SPLINE
SPL {X  -120.253, Y  +789.426, Z    +0.000, E1   -51.165, E3 +212498.946}
SPL {X  -143.101, Y  +758.939, Z    +0.000, E1   -44.365, E3 +212513.054}
SPL {X  -158.740, Y  +722.846, Z    +0.000, E1   -30.140, E3 +212511.093}
SPL {X  -163.639, Y  +701.236, Z    +0.000, E1   -18.901, E3 +212513.231}
SPL {X  -165.058, Y  +689.494, Z    +0.000, E1   -11.557, E3 +212512.047}
SPL {X  -165.574, Y  +680.514, Z    +0.000, E1    -5.500, E3 +212511.291}
SPL {X  -165.650, Y  +673.883, Z    +0.000, E1    -0.454, E3 +212510.302}
SPL {X  -165.650, Y  +672.004, Z    +0.000, E1    +1.620, E3 +212509.508}
SPL {X  -165.650, Y  +669.258, Z    +0.000, E1    +5.269, E3 +212509.126}
SPL {X  -165.650, Y  +665.011, Z    +0.000, E1   +11.627, E3 +212509.014}
SPL {X  -165.650, Y  +659.446, Z    +0.000, E1   +21.123, E3 +212507.878}
SPL {X  -165.650, Y  +654.020, Z    +0.000, E1   +29.754, E3 +212508.032}
SPL {X  -165.650, Y  +644.843, Z    +0.000, E1   +43.427, E3 +212506.358}
SPL {X  -165.650, Y  +632.102, Z    +0.000, E1   +56.225, E3 +212505.707}
SPL {X  -165.650, Y  +581.672, Z    +0.000, E1   +69.744, E3 +212518.099}
SPL {X  -165.650, Y  +458.048, Z    +0.000, E1   +68.782, E3 +212598.832}
ENDSPLINE

SPLINE
SPL {X  -165.650, Y  +484.472, Z    +0.000, E1   +63.918, E3 +212613.083}
ENDSPLINE

SPLINE
SPL {X  -165.650, Y  +477.868, Z    +0.000, E1   +63.324, E3 +212624.260}
SPL {X  -165.650, Y  +463.578, Z    +0.000, E1   +63.625, E3 +212636.614}
SPL {X  -165.650, Y  +453.769, Z    +0.000, E1   +63.450, E3 +212647.873}
SPL {X  -165.650, Y  +444.234, Z    +0.000, E1   +63.262, E3 +212659.046}
SPL {X  -165.650, Y  +432.479, Z    +0.000, E1   +63.557, E3 +212668.866}
SPL {X  -165.650, Y  +422.068, Z    +0.000, E1   +63.630, E3 +212678.961}
SPL {X  -165.650, Y  +411.650, Z    +0.000, E1   +63.439, E3 +212690.979}
SPL {X  -165.650, Y  +399.089, Z    +0.000, E1   +63.334, E3 +212704.705}
ENDSPLINE

SPLINE
SPL {X  -165.650, Y  +410.094, Z    +0.000, E1   +60.049, E3 +212715.422}
ENDSPLINE

SPLINE
SPL {X  -165.650, Y  +398.700, Z    +0.000, E1   +60.415, E3 +212726.320}
SPL {X  -165.650, Y  +380.643, Z    +0.000, E1   +61.187, E3 +212741.682}
SPL {X  -165.125, Y  +365.326, Z    +0.000, E1   +61.696, E3 +212755.025}
SPL {X  -164.823, Y  +361.969, Z    +0.000, E1   +60.899, E3 +212764.260}
SPL {X  -163.414, Y  +351.372, Z    +0.000, E1   +61.284, E3 +212773.522}
SPL {X  -162.189, Y  +344.818, Z    +0.000, E1   +60.900, E3 +212783.376}
SPL {X  -160.769, Y  +338.584, Z    +0.000, E1   +60.413, E3 +212793.552}
SPL {X  -158.568, Y  +330.583, Z    +0.000, E1   +60.533, E3 +212801.692}
SPL {X  -157.003, Y  +325.679, Z    +0.000, E1   +60.284, E3 +212808.662}
SPL {X  -155.286, Y  +320.826, Z    +0.000, E1   +59.686, E3 +212817.774}
SPL {X  -151.657, Y  +311.865, Z    +0.000, E1   +59.311, E3 +212830.076}
SPL {X  -147.428, Y  +302.969, Z    +0.000, E1   +58.548, E3 +212844.092}
SPL {X  -143.281, Y  +295.370, Z    +0.000, E1   +57.860, E3 +212855.891}
SPL {X  -136.453, Y  +284.583, Z    +0.000, E1   +60.257, E3 +212856.375}
SPL {X  -128.205, Y  +273.602, Z    +0.000, E1   +62.388, E3 +212857.079}
SPL {X   -93.591, Y  +241.823, Z    +0.000, E1   +55.455, E3 +212949.208}
ENDSPLINE

SPLINE
SPL {X  -110.554, Y  +255.140, Z    +0.000, E1   +52.082, E3 +213076.164}
SPL {X  -137.038, Y  +285.439, Z    +0.000, E1   +46.261, E3 +213095.904}
SPL {X  -149.954, Y  +308.117, Z    +0.000, E1   +39.560, E3 +213102.252}
SPL {X  -160.070, Y  +335.868, Z    +0.000, E1   +27.320, E3 +213096.650}
SPL {X  -163.969, Y  +354.959, Z    +0.000, E1   +17.178, E3 +213097.164}
SPL {X  -165.261, Y  +367.153, Z    +0.000, E1    +9.611, E3 +213096.317}
SPL {X  -165.600, Y  +374.440, Z    +0.000, E1    +4.699, E3 +213095.578}
SPL {X  -165.650, Y  +379.657, Z    +0.000, E1    +0.819, E3 +213095.106}
SPL {X  -165.650, Y  +381.885, Z    +0.000, E1    -1.282, E3 +213094.351}
SPL {X  -165.650, Y  +386.855, Z    +0.000, E1    -7.700, E3 +213093.770}
SPL {X  -165.650, Y  +393.198, Z    +0.000, E1   -17.733, E3 +213092.745}
SPL {X  -165.650, Y  +399.991, Z    +0.000, E1   -27.922, E3 +213093.641}
SPL {X  -165.650, Y  +409.148, Z    +0.000, E1   -43.235, E3 +213089.028}
SPL {X  -165.650, Y  +420.563, Z    +0.000, E1   -54.059, E3 +213089.585}
SPL {X  -165.650, Y  +436.566, Z    +0.000, E1   -62.888, E3 +213091.298}
SPL {X  -165.650, Y  +479.770, Z    +0.000, E1   -67.621, E3 +213110.637}
SPL {X  -165.650, Y  +594.725, Z    +0.000, E1   -69.155, E3 +213178.099}
ENDSPLINE

SPLINE
SPL {X  -165.650, Y  +565.175, Z    +0.000, E1   -62.653, E3 +213201.590}
ENDSPLINE

SPLINE
SPL {X  -165.650, Y  +576.067, Z    +0.000, E1   -62.373, E3 +213214.991}
SPL {X  -165.650, Y  +586.101, Z    +0.000, E1   -62.398, E3 +213225.573}
SPL {X  -165.650, Y  +596.110, Z    +0.000, E1   -62.302, E3 +213237.014}
SPL {X  -165.650, Y  +607.052, Z    +0.000, E1   -62.387, E3 +213248.081}
SPL {X  -165.650, Y  +615.372, Z    +0.000, E1   -62.260, E3 +213257.908}
SPL {X  -165.650, Y  +628.571, Z    +0.000, E1   -62.348, E3 +213271.629}
SPL {X  -165.650, Y  +640.498, Z    +0.000, E1   -62.343, E3 +213284.250}
SPL {X  -165.650, Y  +654.166, Z    +0.000, E1   -62.507, E3 +213297.902}
SPL {X  -165.650, Y  +665.926, Z    +0.000, E1   -62.171, E3 +213312.700}
SPL {X  -165.600, Y  +679.566, Z    +0.000, E1   -62.408, E3 +213325.737}
SPL {X  -165.066, Y  +689.394, Z    +0.000, E1   -62.143, E3 +213338.067}
SPL {X  -164.056, Y  +698.425, Z    +0.000, E1   -62.113, E3 +213347.987}
SPL {X  -162.891, Y  +705.608, Z    +0.000, E1   -61.899, E3 +213357.158}
SPL {X  -160.709, Y  +715.657, Z    +0.000, E1   -61.639, E3 +213369.910}
SPL {X  -157.706, Y  +726.183, Z    +0.000, E1   -61.153, E3 +213384.293}
SPL {X  -155.057, Y  +733.785, Z    +0.000, E1   -60.834, E3 +213394.283}
SPL {X  -152.882, Y  +739.274, Z    +0.000, E1   -60.485, E3 +213402.275}
SPL {X  -150.387, Y  +744.953, Z    +0.000, E1   -60.023, E3 +213410.950}
SPL {X  -146.839, Y  +752.170, Z    +0.000, E1   -59.458, E3 +213421.909}
SPL {X  -142.415, Y  +760.104, Z    +0.000, E1   -58.730, E3 +213433.968}
SPL {X  -132.386, Y  +775.068, Z    +0.000, E1   -61.559, E3 +213436.037}
SPL {X   -89.692, Y  +814.767, Z    +0.000, E1   -54.641, E3 +213550.086}
ENDSPLINE

SPLINE
SPL {X  -133.336, Y  +773.792, Z    +0.000, E1   -47.991, E3 +213678.553}
SPL {X  -153.017, Y  +738.949, Z    +0.000, E1   -37.928, E3 +213691.957}
SPL {X  -160.146, Y  +717.846, Z    +0.000, E1   -27.412, E3 +213679.503}
SPL {X  -163.639, Y  +701.236, Z    +0.000, E1   -18.901, E3 +213685.644}
SPL {X  -165.058, Y  +689.494, Z    +0.000, E1   -11.557, E3 +213684.461}
SPL {X  -165.574, Y  +680.514, Z    +0.000, E1    -5.500, E3 +213683.705}
SPL {X  -165.650, Y  +673.883, Z    +0.000, E1    -0.454, E3 +213682.716}
SPL {X  -165.650, Y  +672.004, Z    +0.000, E1    +1.620, E3 +213681.922}
SPL {X  -165.650, Y  +669.258, Z    +0.000, E1    +5.269, E3 +213681.540}
SPL {X  -165.650, Y  +665.011, Z    +0.000, E1   +11.627, E3 +213681.427}
SPL {X  -165.650, Y  +659.446, Z    +0.000, E1   +21.123, E3 +213680.292}
SPL {X  -165.650, Y  +654.020, Z    +0.000, E1   +29.754, E3 +213680.446}
SPL {X  -165.650, Y  +644.843, Z    +0.000, E1   +43.427, E3 +213678.772}
SPL {X  -165.650, Y  +632.102, Z    +0.000, E1   +56.225, E3 +213678.121}
SPL {X  -165.650, Y  +581.672, Z    +0.000, E1   +69.744, E3 +213690.513}
SPL {X  -165.650, Y  +458.048, Z    +0.000, E1   +68.782, E3 +213771.246}
ENDSPLINE

SPLINE
SPL {X  -165.650, Y  +484.472, Z    +0.000, E1   +63.918, E3 +213785.496}
ENDSPLINE

SPLINE
SPL {X  -165.650, Y  +477.868, Z    +0.000, E1   +63.324, E3 +213796.674}
SPL {X  -165.650, Y  +463.578, Z    +0.000, E1   +63.625, E3 +213809.028}
SPL {X  -165.650, Y  +453.769, Z    +0.000, E1   +63.450, E3 +213820.286}
SPL {X  -165.650, Y  +444.234, Z    +0.000, E1   +63.262, E3 +213831.459}
SPL {X  -165.650, Y  +432.479, Z    +0.000, E1   +63.557, E3 +213841.279}
SPL {X  -165.650, Y  +422.068, Z    +0.000, E1   +63.630, E3 +213851.375}
SPL {X  -165.650, Y  +411.650, Z    +0.000, E1   +63.439, E3 +213863.393}
SPL {X  -165.650, Y  +399.089, Z    +0.000, E1   +63.334, E3 +213877.118}
ENDSPLINE

SPLINE
SPL {X  -165.650, Y  +410.094, Z    +0.000, E1   +60.049, E3 +213887.836}
ENDSPLINE

SPLINE
SPL {X  -165.650, Y  +398.700, Z    +0.000, E1   +60.415, E3 +213898.734}
SPL {X  -165.650, Y  +380.643, Z    +0.000, E1   +61.187, E3 +213914.095}
SPL {X  -165.125, Y  +365.326, Z    +0.000, E1   +61.696, E3 +213927.439}
SPL {X  -164.823, Y  +361.969, Z    +0.000, E1   +60.899, E3 +213936.674}
SPL {X  -163.414, Y  +351.372, Z    +0.000, E1   +61.284, E3 +213945.936}
SPL {X  -162.189, Y  +344.818, Z    +0.000, E1   +60.900, E3 +213955.790}
SPL {X  -160.769, Y  +338.584, Z    +0.000, E1   +60.413, E3 +213965.965}
SPL {X  -157.780, Y  +328.049, Z    +0.000, E1   +60.445, E3 +213977.632}
SPL {X  -155.286, Y  +320.826, Z    +0.000, E1   +59.686, E3 +213990.188}
SPL {X  -152.445, Y  +313.689, Z    +0.000, E1   +59.490, E3 +213999.253}
SPL {X  -150.678, Y  +309.680, Z    +0.000, E1   +58.971, E3 +214006.565}
SPL {X  -148.010, Y  +304.117, Z    +0.000, E1   +58.696, E3 +214014.312}
SPL {X  -144.822, Y  +298.086, Z    +0.000, E1   +58.093, E3 +214024.094}
SPL {X  -142.530, Y  +294.089, Z    +0.000, E1   +57.567, E3 +214030.978}
SPL {X  -134.010, Y  +281.128, Z    +0.000, E1   +60.923, E3 +214029.084}
SPL {X   -93.591, Y  +241.823, Z    +0.000, E1   +55.455, E3 +214121.622}
ENDSPLINE

SPLINE
SPL {X  -110.554, Y  +255.140, Z    +0.000, E1   +52.082, E3 +214248.578}
SPL {X  -144.988, Y  +298.385, Z    +0.000, E1   +42.755, E3 +214272.397}
SPL {X  -160.070, Y  +335.868, Z    +0.000, E1   +27.320, E3 +214269.064}
SPL {X  -163.969, Y  +354.959, Z    +0.000, E1   +17.178, E3 +214269.578}
SPL {X  -165.261, Y  +367.153, Z    +0.000, E1    +9.611, E3 +214268.731}
SPL {X  -165.600, Y  +374.440, Z    +0.000, E1    +4.699, E3 +214267.992}
SPL {X  -165.650, Y  +380.303, Z    +0.000, E1    +0.337, E3 +214267.202}
SPL {X  -165.650, Y  +382.684, Z    +0.000, E1    -2.314, E3 +214266.697}
SPL {X  -165.650, Y  +385.555, Z    +0.000, E1    -6.051, E3 +214265.910}
SPL {X  -165.650, Y  +388.884, Z    +0.000, E1   -10.835, E3 +214266.610}
SPL {X  -165.650, Y  +393.198, Z    +0.000, E1   -17.733, E3 +214265.159}
SPL {X  -165.650, Y  +399.991, Z    +0.000, E1   -27.922, E3 +214266.055}
SPL {X  -165.650, Y  +409.148, Z    +0.000, E1   -43.235, E3 +214261.441}
SPL {X  -165.650, Y  +420.563, Z    +0.000, E1   -54.059, E3 +214261.999}
SPL {X  -165.650, Y  +436.566, Z    +0.000, E1   -62.888, E3 +214263.712}
SPL {X  -165.650, Y  +479.770, Z    +0.000, E1   -67.621, E3 +214283.051}
SPL {X  -165.650, Y  +594.725, Z    +0.000, E1   -69.155, E3 +214350.513}
ENDSPLINE

SPLINE
SPL {X  -165.650, Y  +562.482, Z    +0.000, E1   -62.785, E3 +214369.978}
ENDSPLINE

SPLINE
SPL {X  -165.650, Y  +572.898, Z    +0.000, E1   -62.409, E3 +214383.916}
SPL {X  -165.650, Y  +586.101, Z    +0.000, E1   -62.398, E3 +214397.987}
SPL {X  -165.650, Y  +596.110, Z    +0.000, E1   -62.302, E3 +214409.428}
SPL {X  -165.650, Y  +607.052, Z    +0.000, E1   -62.387, E3 +214420.495}
SPL {X  -165.650, Y  +615.372, Z    +0.000, E1   -62.260, E3 +214430.322}
SPL {X  -165.650, Y  +628.571, Z    +0.000, E1   -62.348, E3 +214444.043}
SPL {X  -165.650, Y  +645.288, Z    +0.000, E1   -62.475, E3 +214460.982}
SPL {X  -165.650, Y  +657.265, Z    +0.000, E1   -62.410, E3 +214474.100}
SPL {X  -165.650, Y  +665.926, Z    +0.000, E1   -62.171, E3 +214485.114}
SPL {X  -165.600, Y  +679.566, Z    +0.000, E1   -62.408, E3 +214498.151}
SPL {X  -165.066, Y  +689.394, Z    +0.000, E1   -62.143, E3 +214510.480}
SPL {X  -164.056, Y  +698.425, Z    +0.000, E1   -62.113, E3 +214520.401}
SPL {X  -162.891, Y  +705.608, Z    +0.000, E1   -61.899, E3 +214529.572}
SPL {X  -160.709, Y  +715.657, Z    +0.000, E1   -61.639, E3 +214542.324}
SPL {X  -157.706, Y  +726.183, Z    +0.000, E1   -61.153, E3 +214556.707}
SPL {X  -155.057, Y  +733.785, Z    +0.000, E1   -60.834, E3 +214566.697}
SPL {X  -152.882, Y  +739.274, Z    +0.000, E1   -60.485, E3 +214574.689}
SPL {X  -149.755, Y  +746.304, Z    +0.000, E1   -59.867, E3 +214585.811}
SPL {X  -146.068, Y  +753.629, Z    +0.000, E1   -59.384, E3 +214596.170}
SPL {X  -143.119, Y  +758.908, Z    +0.000, E1   -58.828, E3 +214604.544}
SPL {X  -141.017, Y  +762.414, Z    +0.000, E1   -58.435, E3 +214610.065}
SPL {X  -132.386, Y  +775.068, Z    +0.000, E1   -61.559, E3 +214608.450}
SPL {X   -89.692, Y  +814.767, Z    +0.000, E1   -54.641, E3 +214722.500}
ENDSPLINE

SPLINE
SPL {X  -133.336, Y  +773.792, Z    +0.000, E1   -47.991, E3 +214850.967}
SPL {X  -153.017, Y  +738.949, Z    +0.000, E1   -37.928, E3 +214864.370}
SPL {X  -160.146, Y  +717.846, Z    +0.000, E1   -27.412, E3 +214851.917}
SPL {X  -163.639, Y  +701.236, Z    +0.000, E1   -18.901, E3 +214858.058}
SPL {X  -165.058, Y  +689.494, Z    +0.000, E1   -11.557, E3 +214856.875}
SPL {X  -165.574, Y  +680.514, Z    +0.000, E1    -5.500, E3 +214856.119}
SPL {X  -165.650, Y  +674.881, Z    +0.000, E1    -1.215, E3 +214855.722}
SPL {X  -165.650, Y  +673.425, Z    +0.000, E1    +0.051, E3 +214854.857}
SPL {X  -165.650, Y  +672.004, Z    +0.000, E1    +1.620, E3 +214854.336}
SPL {X  -165.650, Y  +669.258, Z    +0.000, E1    +5.269, E3 +214853.954}
SPL {X  -165.650, Y  +665.011, Z    +0.000, E1   +11.627, E3 +214853.841}
SPL {X  -165.650, Y  +659.446, Z    +0.000, E1   +21.123, E3 +214852.705}
SPL {X  -165.650, Y  +651.038, Z    +0.000, E1   +34.281, E3 +214852.331}
SPL {X  -165.650, Y  +635.255, Z    +0.000, E1   +53.641, E3 +214850.519}
SPL {X  -165.650, Y  +581.672, Z    +0.000, E1   +69.744, E3 +214862.927}
SPL {X  -165.650, Y  +458.048, Z    +0.000, E1   +68.782, E3 +214943.660}
ENDSPLINE

SPLINE
SPL {X  -165.650, Y  +484.472, Z    +0.000, E1   +63.918, E3 +214957.910}
ENDSPLINE

SPLINE
SPL {X  -165.650, Y  +477.868, Z    +0.000, E1   +63.324, E3 +214969.088}
SPL {X  -165.650, Y  +463.578, Z    +0.000, E1   +63.625, E3 +214981.442}
SPL {X  -165.650, Y  +453.769, Z    +0.000, E1   +63.450, E3 +214992.700}
SPL {X  -165.650, Y  +444.234, Z    +0.000, E1   +63.262, E3 +215003.873}
SPL {X  -165.650, Y  +432.479, Z    +0.000, E1   +63.557, E3 +215013.693}
SPL {X  -165.650, Y  +422.068, Z    +0.000, E1   +63.630, E3 +215023.788}
SPL {X  -165.650, Y  +409.231, Z    +0.000, E1   +63.364, E3 +215039.037}
SPL {X  -165.650, Y  +395.008, Z    +0.000, E1   +63.445, E3 +215052.800}
ENDSPLINE

SPLINE
SPL {X  -165.650, Y  +410.094, Z    +0.000, E1   +60.049, E3 +215060.250}
ENDSPLINE

SPLINE
SPL {X  -165.650, Y  +398.700, Z    +0.000, E1   +60.415, E3 +215071.147}
SPL {X  -165.650, Y  +380.643, Z    +0.000, E1   +61.187, E3 +215086.509}
SPL {X  -165.125, Y  +365.326, Z    +0.000, E1   +61.696, E3 +215099.853}
SPL {X  -164.823, Y  +361.969, Z    +0.000, E1   +60.899, E3 +215109.088}
SPL {X  -163.414, Y  +351.372, Z    +0.000, E1   +61.284, E3 +215118.350}
SPL {X  -162.189, Y  +344.818, Z    +0.000, E1   +60.900, E3 +215128.203}
SPL {X  -160.769, Y  +338.584, Z    +0.000, E1   +60.413, E3 +215138.379}
SPL {X  -157.780, Y  +328.049, Z    +0.000, E1   +60.445, E3 +215150.046}
SPL {X  -155.286, Y  +320.826, Z    +0.000, E1   +59.686, E3 +215162.602}
SPL {X  -152.445, Y  +313.689, Z    +0.000, E1   +59.490, E3 +215171.667}
SPL {X  -149.851, Y  +307.898, Z    +0.000, E1   +58.978, E3 +215180.989}
SPL {X  -146.926, Y  +301.997, Z    +0.000, E1   +58.334, E3 +215190.951}
SPL {X  -143.281, Y  +295.370, Z    +0.000, E1   +57.860, E3 +215200.719}
SPL {X  -134.010, Y  +281.128, Z    +0.000, E1   +60.923, E3 +215201.498}
SPL {X   -93.591, Y  +241.823, Z    +0.000, E1   +55.455, E3 +215294.036}
ENDSPLINE

SPLINE
SPL {X  -110.554, Y  +255.140, Z    +0.000, E1   +52.082, E3 +215420.992}
SPL {X  -137.038, Y  +285.439, Z    +0.000, E1   +46.261, E3 +215440.731}
SPL {X  -149.954, Y  +308.117, Z    +0.000, E1   +39.560, E3 +215447.079}
SPL {X  -160.070, Y  +335.868, Z    +0.000, E1   +27.320, E3 +215441.478}
SPL {X  -163.969, Y  +354.959, Z    +0.000, E1   +17.178, E3 +215441.992}
SPL {X  -165.261, Y  +367.153, Z    +0.000, E1    +9.611, E3 +215441.144}
SPL {X  -165.600, Y  +374.440, Z    +0.000, E1    +4.699, E3 +215440.406}
SPL {X  -165.650, Y  +380.303, Z    +0.000, E1    +0.337, E3 +215439.616}
SPL {X  -165.650, Y  +382.684, Z    +0.000, E1    -2.314, E3 +215439.110}
SPL {X  -165.650, Y  +386.855, Z    +0.000, E1    -7.700, E3 +215438.597}
SPL {X  -165.650, Y  +393.198, Z    +0.000, E1   -17.733, E3 +215437.573}
SPL {X  -165.650, Y  +399.991, Z    +0.000, E1   -27.922, E3 +215438.469}
SPL {X  -165.650, Y  +409.148, Z    +0.000, E1   -43.235, E3 +215433.855}
SPL {X  -165.650, Y  +420.563, Z    +0.000, E1   -54.059, E3 +215434.413}
SPL {X  -165.650, Y  +436.566, Z    +0.000, E1   -62.888, E3 +215436.126}
SPL {X  -165.650, Y  +479.770, Z    +0.000, E1   -67.621, E3 +215455.465}
SPL {X  -165.650, Y  +594.725, Z    +0.000, E1   -69.155, E3 +215522.927}
ENDSPLINE

SPLINE
SPL {X  -165.650, Y  +565.175, Z    +0.000, E1   -62.653, E3 +215546.417}
ENDSPLINE

SPLINE
SPL {X  -165.650, Y  +576.067, Z    +0.000, E1   -62.373, E3 +215559.819}
SPL {X  -165.650, Y  +586.101, Z    +0.000, E1   -62.398, E3 +215570.401}
SPL {X  -165.650, Y  +596.110, Z    +0.000, E1   -62.302, E3 +215581.841}
SPL {X  -165.650, Y  +607.052, Z    +0.000, E1   -62.387, E3 +215592.909}
SPL {X  -165.650, Y  +618.920, Z    +0.000, E1   -62.340, E3 +215606.099}
SPL {X  -165.650, Y  +631.247, Z    +0.000, E1   -62.270, E3 +215619.715}
SPL {X  -165.650, Y  +645.288, Z    +0.000, E1   -62.475, E3 +215633.396}
SPL {X  -165.650, Y  +657.265, Z    +0.000, E1   -62.410, E3 +215646.514}
SPL {X  -165.650, Y  +665.926, Z    +0.000, E1   -62.171, E3 +215657.528}
SPL {X  -165.644, Y  +676.899, Z    +0.000, E1   -62.447, E3 +215667.295}
SPL {X  -165.241, Y  +687.133, Z    +0.000, E1   -62.230, E3 +215679.998}
SPL {X  -164.056, Y  +698.425, Z    +0.000, E1   -62.113, E3 +215692.814}
SPL {X  -162.891, Y  +705.608, Z    +0.000, E1   -61.899, E3 +215701.986}
SPL {X  -160.709, Y  +715.657, Z    +0.000, E1   -61.639, E3 +215714.738}
SPL {X  -157.706, Y  +726.183, Z    +0.000, E1   -61.153, E3 +215729.121}
SPL {X  -155.057, Y  +733.785, Z    +0.000, E1   -60.834, E3 +215739.110}
SPL {X  -152.882, Y  +739.274, Z    +0.000, E1   -60.485, E3 +215747.103}
SPL {X  -150.387, Y  +744.953, Z    +0.000, E1   -60.023, E3 +215755.778}
SPL {X  -146.839, Y  +752.170, Z    +0.000, E1   -59.458, E3 +215766.737}
SPL {X  -142.415, Y  +760.104, Z    +0.000, E1   -58.730, E3 +215778.796}
SPL {X  -132.386, Y  +775.068, Z    +0.000, E1   -61.559, E3 +215780.864}
SPL {X   -89.692, Y  +814.767, Z    +0.000, E1   -54.641, E3 +215894.913}
ENDSPLINE

SPLINE
SPL {X  -133.336, Y  +773.792, Z    +0.000, E1   -47.991, E3 +216023.380}
SPL {X  -153.017, Y  +738.949, Z    +0.000, E1   -37.928, E3 +216036.784}
SPL {X  -160.146, Y  +717.846, Z    +0.000, E1   -27.412, E3 +216024.331}
SPL {X  -163.639, Y  +701.236, Z    +0.000, E1   -18.901, E3 +216030.472}
SPL {X  -165.058, Y  +689.494, Z    +0.000, E1   -11.557, E3 +216029.289}
SPL {X  -165.574, Y  +680.514, Z    +0.000, E1    -5.500, E3 +216028.532}
SPL {X  -165.650, Y  +673.883, Z    +0.000, E1    -0.454, E3 +216027.543}
SPL {X  -165.650, Y  +672.004, Z    +0.000, E1    +1.620, E3 +216026.749}
SPL {X  -165.650, Y  +669.258, Z    +0.000, E1    +5.269, E3 +216026.368}
SPL {X  -165.650, Y  +665.011, Z    +0.000, E1   +11.627, E3 +216026.255}
SPL {X  -165.650, Y  +659.446, Z    +0.000, E1   +21.123, E3 +216025.119}
SPL {X  -165.650, Y  +654.020, Z    +0.000, E1   +29.754, E3 +216025.274}
SPL {X  -165.650, Y  +644.843, Z    +0.000, E1   +43.427, E3 +216023.600}
SPL {X  -165.650, Y  +632.102, Z    +0.000, E1   +56.225, E3 +216022.948}
SPL {X  -165.650, Y  +581.672, Z    +0.000, E1   +69.744, E3 +216035.341}
SPL {X  -165.650, Y  +458.048, Z    +0.000, E1   +68.782, E3 +216116.073}
ENDSPLINE

SPLINE
SPL {X  -165.650, Y  +484.472, Z    +0.000, E1   +63.918, E3 +216130.324}
ENDSPLINE

SPLINE
SPL {X  -165.650, Y  +477.868, Z    +0.000, E1   +63.324, E3 +216141.502}
SPL {X  -165.650, Y  +463.578, Z    +0.000, E1   +63.625, E3 +216153.855}
SPL {X  -165.650, Y  +453.769, Z    +0.000, E1   +63.450, E3 +216165.114}
SPL {X  -165.650, Y  +444.234, Z    +0.000, E1   +63.262, E3 +216176.287}
SPL {X  -165.650, Y  +432.479, Z    +0.000, E1   +63.557, E3 +216186.107}
SPL {X  -165.650, Y  +422.068, Z    +0.000, E1   +63.630, E3 +216196.202}
SPL {X  -165.650, Y  +411.650, Z    +0.000, E1   +63.439, E3 +216208.221}
SPL {X  -165.650, Y  +399.089, Z    +0.000, E1   +63.334, E3 +216221.946}
ENDSPLINE

SPLINE
SPL {X  -165.650, Y  +410.094, Z    +0.000, E1   +60.049, E3 +216232.663}
ENDSPLINE

SPLINE
SPL {X  -165.650, Y  +398.700, Z    +0.000, E1   +60.415, E3 +216243.561}
SPL {X  -165.650, Y  +382.616, Z    +0.000, E1   +61.427, E3 +216254.780}
SPL {X  -165.650, Y  +379.013, Z    +0.000, E1   +60.888, E3 +216262.602}
SPL {X  -165.125, Y  +365.326, Z    +0.000, E1   +61.696, E3 +216272.266}
SPL {X  -164.823, Y  +361.969, Z    +0.000, E1   +60.899, E3 +216281.501}
SPL {X  -163.414, Y  +351.372, Z    +0.000, E1   +61.284, E3 +216290.764}
SPL {X  -162.189, Y  +344.818, Z    +0.000, E1   +60.900, E3 +216300.617}
SPL {X  -160.769, Y  +338.584, Z    +0.000, E1   +60.413, E3 +216310.793}
SPL {X  -157.780, Y  +328.049, Z    +0.000, E1   +60.445, E3 +216322.460}
SPL {X  -155.286, Y  +320.826, Z    +0.000, E1   +59.686, E3 +216335.015}
SPL {X  -152.445, Y  +313.689, Z    +0.000, E1   +59.490, E3 +216344.081}
SPL {X  -149.851, Y  +307.898, Z    +0.000, E1   +58.978, E3 +216353.403}
SPL {X  -146.926, Y  +301.997, Z    +0.000, E1   +58.334, E3 +216363.364}
SPL {X  -143.997, Y  +296.618, Z    +0.000, E1   +58.069, E3 +216370.623}
SPL {X  -142.530, Y  +294.089, Z    +0.000, E1   +57.567, E3 +216375.806}
SPL {X  -134.010, Y  +281.128, Z    +0.000, E1   +60.923, E3 +216373.911}
SPL {X   -93.591, Y  +241.823, Z    +0.000, E1   +55.455, E3 +216466.449}
ENDSPLINE

SPLINE
SPL {X  -110.554, Y  +255.140, Z    +0.000, E1   +52.082, E3 +216593.406}
SPL {X  -137.038, Y  +285.439, Z    +0.000, E1   +46.261, E3 +216613.145}
SPL {X  -149.954, Y  +308.117, Z    +0.000, E1   +39.560, E3 +216619.493}
SPL {X  -160.070, Y  +335.868, Z    +0.000, E1   +27.320, E3 +216613.892}
SPL {X  -163.969, Y  +354.959, Z    +0.000, E1   +17.178, E3 +216614.406}
SPL {X  -165.261, Y  +367.153, Z    +0.000, E1    +9.611, E3 +216613.558}
SPL {X  -165.600, Y  +374.440, Z    +0.000, E1    +4.699, E3 +216612.819}
SPL {X  -165.650, Y  +379.657, Z    +0.000, E1    +0.819, E3 +216612.348}
SPL {X  -165.650, Y  +381.885, Z    +0.000, E1    -1.282, E3 +216611.592}
SPL {X  -165.650, Y  +386.855, Z    +0.000, E1    -7.700, E3 +216611.011}
SPL {X  -165.650, Y  +393.198, Z    +0.000, E1   -17.733, E3 +216609.987}
SPL {X  -165.650, Y  +399.991, Z    +0.000, E1   -27.922, E3 +216610.883}
SPL {X  -165.650, Y  +411.457, Z    +0.000, E1   -45.557, E3 +216606.630}
SPL {X  -165.650, Y  +427.627, Z    +0.000, E1   -58.747, E3 +216607.264}
SPL {X  -165.650, Y  +479.770, Z    +0.000, E1   -67.621, E3 +216627.879}
SPL {X  -165.650, Y  +594.725, Z    +0.000, E1   -69.155, E3 +216695.340}
ENDSPLINE

SPLINE
SPL {X  -165.650, Y  +565.175, Z    +0.000, E1   -62.653, E3 +216718.831}
ENDSPLINE

SPLINE
SPL {X  -165.650, Y  +576.067, Z    +0.000, E1   -62.373, E3 +216732.232}
SPL {X  -165.650, Y  +586.101, Z    +0.000, E1   -62.398, E3 +216742.814}
SPL {X  -165.650, Y  +596.110, Z    +0.000, E1   -62.302, E3 +216754.255}
SPL {X  -165.650, Y  +607.052, Z    +0.000, E1   -62.387, E3 +216765.322}
SPL {X  -165.650, Y  +615.372, Z    +0.000, E1   -62.260, E3 +216775.150}
SPL {X  -165.650, Y  +628.571, Z    +0.000, E1   -62.348, E3 +216788.870}
SPL {X  -165.650, Y  +640.498, Z    +0.000, E1   -62.343, E3 +216801.492}
SPL {X  -165.650, Y  +654.166, Z    +0.000, E1   -62.507, E3 +216815.143}
SPL {X  -165.650, Y  +665.926, Z    +0.000, E1   -62.171, E3 +216829.941}
SPL {X  -165.600, Y  +679.566, Z    +0.000, E1   -62.408, E3 +216842.979}
SPL {X  -165.066, Y  +689.394, Z    +0.000, E1   -62.143, E3 +216855.308}
SPL {X  -164.056, Y  +698.425, Z    +0.000, E1   -62.113, E3 +216865.228}
SPL {X  -162.891, Y  +705.608, Z    +0.000, E1   -61.899, E3 +216874.400}
SPL {X  -161.308, Y  +713.180, Z    +0.000, E1   -61.813, E3 +216883.093}
SPL {X  -159.339, Y  +720.787, Z    +0.000, E1   -61.452, E3 +216893.789}
SPL {X  -156.103, Y  +730.922, Z    +0.000, E1   -60.875, E3 +216908.335}
SPL {X  -152.882, Y  +739.274, Z    +0.000, E1   -60.485, E3 +216919.517}
SPL {X  -149.755, Y  +746.304, Z    +0.000, E1   -59.867, E3 +216930.638}
SPL {X  -146.068, Y  +753.629, Z    +0.000, E1   -59.384, E3 +216940.997}
SPL {X  -142.415, Y  +760.104, Z    +0.000, E1   -58.730, E3 +216951.209}
SPL {X  -132.386, Y  +775.068, Z    +0.000, E1   -61.559, E3 +216953.278}
SPL {X   -89.692, Y  +814.767, Z    +0.000, E1   -54.641, E3 +217067.327}
ENDSPLINE

SPLINE
SPL {X  -133.336, Y  +773.792, Z    +0.000, E1   -47.991, E3 +217195.794}
SPL {X  -153.017, Y  +738.949, Z    +0.000, E1   -37.928, E3 +217209.198}
SPL {X  -160.146, Y  +717.846, Z    +0.000, E1   -27.412, E3 +217196.744}
SPL {X  -163.639, Y  +701.236, Z    +0.000, E1   -18.901, E3 +217202.886}
SPL {X  -165.058, Y  +689.494, Z    +0.000, E1   -11.557, E3 +217201.703}
SPL {X  -165.574, Y  +680.514, Z    +0.000, E1    -5.500, E3 +217200.946}
SPL {X  -165.650, Y  +673.883, Z    +0.000, E1    -0.454, E3 +217199.957}
SPL {X  -165.650, Y  +672.004, Z    +0.000, E1    +1.620, E3 +217199.163}
SPL {X  -165.650, Y  +669.258, Z    +0.000, E1    +5.269, E3 +217198.782}
SPL {X  -165.650, Y  +665.011, Z    +0.000, E1   +11.627, E3 +217198.669}
SPL {X  -165.650, Y  +659.446, Z    +0.000, E1   +21.123, E3 +217197.533}
SPL {X  -165.650, Y  +654.020, Z    +0.000, E1   +29.754, E3 +217197.687}
SPL {X  -165.650, Y  +644.843, Z    +0.000, E1   +43.427, E3 +217196.013}
SPL {X  -165.650, Y  +632.102, Z    +0.000, E1   +56.225, E3 +217195.362}
SPL {X  -165.650, Y  +581.672, Z    +0.000, E1   +69.744, E3 +217207.754}
SPL {X  -165.650, Y  +458.048, Z    +0.000, E1   +68.782, E3 +217288.487}
ENDSPLINE

SPLINE
SPL {X  -165.650, Y  +484.472, Z    +0.000, E1   +63.918, E3 +217302.738}
ENDSPLINE

SPLINE
SPL {X  -165.650, Y  +477.868, Z    +0.000, E1   +63.324, E3 +217313.915}
SPL {X  -165.650, Y  +463.578, Z    +0.000, E1   +63.625, E3 +217326.269}
SPL {X  -165.650, Y  +453.769, Z    +0.000, E1   +63.450, E3 +217337.528}
SPL {X  -165.650, Y  +444.234, Z    +0.000, E1   +63.262, E3 +217348.701}
SPL {X  -165.650, Y  +432.479, Z    +0.000, E1   +63.557, E3 +217358.521}
SPL {X  -165.650, Y  +422.068, Z    +0.000, E1   +63.630, E3 +217368.616}
SPL {X  -165.650, Y  +409.231, Z    +0.000, E1   +63.364, E3 +217383.864}
SPL {X  -165.650, Y  +395.008, Z    +0.000, E1   +63.445, E3 +217397.628}
ENDSPLINE

SPLINE
SPL {X  -165.650, Y  +410.094, Z    +0.000, E1   +60.049, E3 +217405.077}
ENDSPLINE

SPLINE
SPL {X  -165.650, Y  +398.700, Z    +0.000, E1   +60.415, E3 +217415.975}
SPL {X  -165.650, Y  +380.643, Z    +0.000, E1   +61.187, E3 +217431.337}
SPL {X  -165.125, Y  +365.326, Z    +0.000, E1   +61.696, E3 +217444.680}
SPL {X  -164.823, Y  +361.969, Z    +0.000, E1   +60.899, E3 +217453.915}
SPL {X  -163.414, Y  +351.372, Z    +0.000, E1   +61.284, E3 +217463.178}
SPL {X  -162.189, Y  +344.818, Z    +0.000, E1   +60.900, E3 +217473.031}
SPL {X  -160.769, Y  +338.584, Z    +0.000, E1   +60.413, E3 +217483.207}
SPL {X  -157.780, Y  +328.049, Z    +0.000, E1   +60.445, E3 +217494.874}
SPL {X  -155.286, Y  +320.826, Z    +0.000, E1   +59.686, E3 +217507.429}
SPL {X  -152.445, Y  +313.689, Z    +0.000, E1   +59.490, E3 +217516.495}
SPL {X  -149.851, Y  +307.898, Z    +0.000, E1   +58.978, E3 +217525.817}
SPL {X  -146.926, Y  +301.997, Z    +0.000, E1   +58.334, E3 +217535.778}
SPL {X  -143.281, Y  +295.370, Z    +0.000, E1   +57.860, E3 +217545.547}
SPL {X  -134.010, Y  +281.128, Z    +0.000, E1   +60.923, E3 +217546.325}
SPL {X   -93.591, Y  +241.823, Z    +0.000, E1   +55.455, E3 +217638.863}
ENDSPLINE

SPLINE
SPL {X  -110.554, Y  +255.140, Z    +0.000, E1   +52.082, E3 +217765.819}
SPL {X  -137.038, Y  +285.439, Z    +0.000, E1   +46.261, E3 +217785.559}
SPL {X  -149.954, Y  +308.117, Z    +0.000, E1   +39.560, E3 +217791.907}
SPL {X  -160.070, Y  +335.868, Z    +0.000, E1   +27.320, E3 +217786.305}
SPL {X  -163.969, Y  +354.959, Z    +0.000, E1   +17.178, E3 +217786.819}
SPL {X  -165.261, Y  +367.153, Z    +0.000, E1    +9.611, E3 +217785.972}
SPL {X  -165.600, Y  +374.440, Z    +0.000, E1    +4.699, E3 +217785.233}
SPL {X  -165.650, Y  +380.303, Z    +0.000, E1    +0.337, E3 +217784.444}
SPL {X  -165.650, Y  +382.684, Z    +0.000, E1    -2.314, E3 +217783.938}
SPL {X  -165.650, Y  +385.555, Z    +0.000, E1    -6.051, E3 +217783.151}
SPL {X  -165.650, Y  +388.884, Z    +0.000, E1   -10.835, E3 +217783.851}
SPL {X  -165.650, Y  +393.198, Z    +0.000, E1   -17.733, E3 +217782.401}
SPL {X  -165.650, Y  +399.991, Z    +0.000, E1   -27.922, E3 +217783.296}
SPL {X  -165.650, Y  +409.148, Z    +0.000, E1   -43.235, E3 +217778.683}
SPL {X  -165.650, Y  +420.563, Z    +0.000, E1   -54.059, E3 +217779.241}
SPL {X  -165.650, Y  +436.566, Z    +0.000, E1   -62.888, E3 +217780.953}
SPL {X  -165.650, Y  +479.770, Z    +0.000, E1   -67.621, E3 +217800.292}
SPL {X  -165.650, Y  +594.725, Z    +0.000, E1   -69.155, E3 +217867.754}
ENDSPLINE

SPLINE
SPL {X  -165.650, Y  +565.175, Z    +0.000, E1   -62.653, E3 +217891.245}
ENDSPLINE

SPLINE
SPL {X  -165.650, Y  +576.067, Z    +0.000, E1   -62.373, E3 +217904.646}
SPL {X  -165.650, Y  +586.101, Z    +0.000, E1   -62.398, E3 +217915.228}
SPL {X  -165.650, Y  +596.110, Z    +0.000, E1   -62.302, E3 +217926.669}
SPL {X  -165.650, Y  +607.052, Z    +0.000, E1   -62.387, E3 +217937.736}
SPL {X  -165.650, Y  +618.920, Z    +0.000, E1   -62.340, E3 +217950.926}
SPL {X  -165.650, Y  +635.445, Z    +0.000, E1   -62.341, E3 +217968.727}
SPL {X  -165.650, Y  +654.166, Z    +0.000, E1   -62.507, E3 +217987.557}
SPL {X  -165.650, Y  +665.926, Z    +0.000, E1   -62.171, E3 +218002.355}
SPL {X  -165.644, Y  +676.899, Z    +0.000, E1   -62.447, E3 +218012.123}
SPL {X  -165.241, Y  +687.133, Z    +0.000, E1   -62.230, E3 +218024.825}
SPL {X  -164.056, Y  +698.425, Z    +0.000, E1   -62.113, E3 +218037.642}
SPL {X  -162.891, Y  +705.608, Z    +0.000, E1   -61.899, E3 +218046.814}
SPL {X  -160.709, Y  +715.657, Z    +0.000, E1   -61.639, E3 +218059.565}
SPL {X  -157.706, Y  +726.183, Z    +0.000, E1   -61.153, E3 +218073.948}
SPL {X  -155.057, Y  +733.785, Z    +0.000, E1   -60.834, E3 +218083.938}
SPL {X  -152.882, Y  +739.274, Z    +0.000, E1   -60.485, E3 +218091.931}
SPL {X  -150.387, Y  +744.953, Z    +0.000, E1   -60.023, E3 +218100.605}
SPL {X  -147.728, Y  +750.443, Z    +0.000, E1   -59.568, E3 +218108.990}
SPL {X  -143.895, Y  +757.561, Z    +0.000, E1   -58.980, E3 +218119.726}
SPL {X  -141.017, Y  +762.414, Z    +0.000, E1   -58.435, E3 +218127.306}
SPL {X  -134.606, Y  +772.046, Z    +0.000, E1   -61.105, E3 +218124.953}
SPL {X  -127.075, Y  +781.763, Z    +0.000, E1   -62.555, E3 +218127.267}
SPL {X   -89.692, Y  +814.767, Z    +0.000, E1   -54.641, E3 +218239.741}
ENDSPLINE

SPLINE
SPL {X  -133.336, Y  +773.792, Z    +0.000, E1   -47.991, E3 +218368.208}
SPL {X  -153.017, Y  +738.949, Z    +0.000, E1   -37.928, E3 +218381.612}
SPL {X  -160.146, Y  +717.846, Z    +0.000, E1   -27.412, E3 +218369.158}
SPL {X  -163.639, Y  +701.236, Z    +0.000, E1   -18.901, E3 +218375.300}
SPL {X  -165.380, Y  +684.951, Z    +0.000, E1    -8.606, E3 +218373.557}
SPL {X  -165.650, Y  +675.640, Z    +0.000, E1    -1.874, E3 +218373.093}
SPL {X  -165.650, Y  +672.727, Z    +0.000, E1    +0.658, E3 +218371.843}
SPL {X  -165.650, Y  +669.258, Z    +0.000, E1    +5.269, E3 +218371.195}
SPL {X  -165.650, Y  +665.011, Z    +0.000, E1   +11.627, E3 +218371.083}
SPL {X  -165.650, Y  +659.446, Z    +0.000, E1   +21.123, E3 +218369.947}
SPL {X  -165.650, Y  +654.020, Z    +0.000, E1   +29.754, E3 +218370.101}
SPL {X  -165.650, Y  +644.843, Z    +0.000, E1   +43.427, E3 +218368.427}
SPL {X  -165.650, Y  +632.102, Z    +0.000, E1   +56.225, E3 +218367.776}
SPL {X  -165.650, Y  +581.672, Z    +0.000, E1   +69.744, E3 +218380.168}
SPL {X  -165.650, Y  +455.882, Z    +0.000, E1   +70.075, E3 +218452.433}
ENDSPLINE

SPLINE
SPL {X  -165.650, Y  +480.501, Z    +0.000, E1   +64.561, E3 +218474.402}
ENDSPLINE

SPLINE
SPL {X  -165.650, Y  +477.868, Z    +0.000, E1   +63.324, E3 +218486.329}
SPL {X  -165.650, Y  +463.578, Z    +0.000, E1   +63.625, E3 +218498.683}
SPL {X  -165.650, Y  +453.769, Z    +0.000, E1   +63.450, E3 +218509.942}
SPL {X  -165.650, Y  +444.234, Z    +0.000, E1   +63.262, E3 +218521.114}
SPL {X  -165.650, Y  +432.479, Z    +0.000, E1   +63.557, E3 +218530.934}
SPL {X  -165.650, Y  +422.068, Z    +0.000, E1   +63.630, E3 +218541.030}
SPL {X  -165.650, Y  +409.231, Z    +0.000, E1   +63.364, E3 +218556.278}
SPL {X  -165.650, Y  +395.008, Z    +0.000, E1   +63.445, E3 +218570.042}
ENDSPLINE

SPLINE
SPL {X  -165.650, Y  +410.094, Z    +0.000, E1   +60.049, E3 +218577.491}
ENDSPLINE

SPLINE
SPL {X  -165.650, Y  +398.700, Z    +0.000, E1   +60.415, E3 +218588.389}
SPL {X  -165.650, Y  +380.643, Z    +0.000, E1   +61.187, E3 +218603.751}
SPL {X  -165.125, Y  +365.326, Z    +0.000, E1   +61.696, E3 +218617.094}
SPL {X  -164.823, Y  +361.969, Z    +0.000, E1   +60.899, E3 +218626.329}
SPL {X  -163.414, Y  +351.372, Z    +0.000, E1   +61.284, E3 +218635.591}
SPL {X  -162.189, Y  +344.818, Z    +0.000, E1   +60.900, E3 +218645.445}
SPL {X  -160.769, Y  +338.584, Z    +0.000, E1   +60.413, E3 +218655.621}
SPL {X  -157.780, Y  +328.049, Z    +0.000, E1   +60.445, E3 +218667.288}
SPL {X  -155.286, Y  +320.826, Z    +0.000, E1   +59.686, E3 +218679.843}
SPL {X  -152.445, Y  +313.689, Z    +0.000, E1   +59.490, E3 +218688.908}
SPL {X  -149.851, Y  +307.898, Z    +0.000, E1   +58.978, E3 +218698.231}
SPL {X  -146.926, Y  +301.997, Z    +0.000, E1   +58.334, E3 +218708.192}
SPL {X  -143.281, Y  +295.370, Z    +0.000, E1   +57.860, E3 +218717.960}
SPL {X  -134.010, Y  +281.128, Z    +0.000, E1   +60.923, E3 +218718.739}
SPL {X   -93.591, Y  +241.823, Z    +0.000, E1   +55.455, E3 +218811.277}
ENDSPLINE

SPLINE
SPL {X  -110.554, Y  +255.140, Z    +0.000, E1   +52.082, E3 +218938.233}
SPL {X  -137.038, Y  +285.439, Z    +0.000, E1   +46.261, E3 +218957.973}
SPL {X  -149.954, Y  +308.117, Z    +0.000, E1   +39.560, E3 +218964.321}
SPL {X  -160.070, Y  +335.868, Z    +0.000, E1   +27.320, E3 +218958.719}
SPL {X  -163.969, Y  +354.959, Z    +0.000, E1   +17.178, E3 +218959.233}
SPL {X  -165.261, Y  +367.153, Z    +0.000, E1    +9.611, E3 +218958.386}
SPL {X  -165.600, Y  +374.440, Z    +0.000, E1    +4.699, E3 +218957.647}
SPL {X  -165.650, Y  +379.657, Z    +0.000, E1    +0.819, E3 +218957.175}
SPL {X  -165.650, Y  +381.885, Z    +0.000, E1    -1.282, E3 +218956.419}
SPL {X  -165.650, Y  +386.855, Z    +0.000, E1    -7.700, E3 +218955.839}
SPL {X  -165.650, Y  +393.198, Z    +0.000, E1   -17.733, E3 +218954.814}
SPL {X  -165.650, Y  +399.991, Z    +0.000, E1   -27.922, E3 +218955.710}
SPL {X  -165.650, Y  +409.148, Z    +0.000, E1   -43.235, E3 +218951.097}
SPL {X  -165.650, Y  +420.563, Z    +0.000, E1   -54.059, E3 +218951.654}
SPL {X  -165.650, Y  +436.566, Z    +0.000, E1   -62.888, E3 +218953.367}
SPL {X  -165.650, Y  +479.770, Z    +0.000, E1   -67.621, E3 +218972.706}
SPL {X  -165.650, Y  +594.725, Z    +0.000, E1   -69.155, E3 +219040.168}
ENDSPLINE

SPLINE
SPL {X  -165.650, Y  +565.175, Z    +0.000, E1   -62.653, E3 +219063.659}
ENDSPLINE

SPLINE
SPL {X  -165.650, Y  +576.067, Z    +0.000, E1   -62.373, E3 +219077.060}
SPL {X  -165.650, Y  +586.101, Z    +0.000, E1   -62.398, E3 +219087.642}
SPL {X  -165.650, Y  +596.110, Z    +0.000, E1   -62.302, E3 +219099.083}
SPL {X  -165.650, Y  +607.052, Z    +0.000, E1   -62.387, E3 +219110.150}
SPL {X  -165.650, Y  +618.920, Z    +0.000, E1   -62.340, E3 +219123.340}
SPL {X  -165.650, Y  +631.247, Z    +0.000, E1   -62.270, E3 +219136.957}
SPL {X  -165.650, Y  +645.288, Z    +0.000, E1   -62.475, E3 +219150.637}
SPL {X  -165.650, Y  +657.265, Z    +0.000, E1   -62.410, E3 +219163.755}
SPL {X  -165.650, Y  +665.926, Z    +0.000, E1   -62.171, E3 +219174.769}
SPL {X  -165.644, Y  +676.899, Z    +0.000, E1   -62.447, E3 +219184.536}
SPL {X  -165.241, Y  +687.133, Z    +0.000, E1   -62.230, E3 +219197.239}
SPL {X  -164.056, Y  +698.425, Z    +0.000, E1   -62.113, E3 +219210.056}
SPL {X  -162.891, Y  +705.608, Z    +0.000, E1   -61.899, E3 +219219.227}
SPL {X  -160.709, Y  +715.657, Z    +0.000, E1   -61.639, E3 +219231.979}
SPL {X  -157.706, Y  +726.183, Z    +0.000, E1   -61.153, E3 +219246.362}
SPL {X  -155.057, Y  +733.785, Z    +0.000, E1   -60.834, E3 +219256.352}
SPL {X  -152.882, Y  +739.274, Z    +0.000, E1   -60.485, E3 +219264.344}
SPL {X  -150.387, Y  +744.953, Z    +0.000, E1   -60.023, E3 +219273.019}
SPL {X  -146.839, Y  +752.170, Z    +0.000, E1   -59.458, E3 +219283.978}
SPL {X  -142.415, Y  +760.104, Z    +0.000, E1   -58.730, E3 +219296.037}
SPL {X  -132.386, Y  +775.068, Z    +0.000, E1   -61.559, E3 +219298.106}
SPL {X   -89.692, Y  +814.767, Z    +0.000, E1   -54.641, E3 +219412.155}
ENDSPLINE

SPLINE
SPL {X  -120.253, Y  +789.426, Z    +0.000, E1   -51.165, E3 +219533.429}
SPL {X  -143.101, Y  +758.939, Z    +0.000, E1   -44.365, E3 +219547.537}
SPL {X  -158.740, Y  +722.846, Z    +0.000, E1   -30.140, E3 +219545.576}
SPL {X  -163.639, Y  +701.236, Z    +0.000, E1   -18.901, E3 +219547.713}
SPL {X  -165.058, Y  +689.494, Z    +0.000, E1   -11.557, E3 +219546.530}
SPL {X  -165.574, Y  +680.514, Z    +0.000, E1    -5.500, E3 +219545.774}
SPL {X  -165.650, Y  +673.883, Z    +0.000, E1    -0.454, E3 +219544.785}
SPL {X  -165.650, Y  +672.004, Z    +0.000, E1    +1.620, E3 +219543.991}
SPL {X  -165.650, Y  +669.258, Z    +0.000, E1    +5.269, E3 +219543.609}
SPL {X  -165.650, Y  +665.011, Z    +0.000, E1   +11.627, E3 +219543.496}
SPL {X  -165.650, Y  +659.446, Z    +0.000, E1   +21.123, E3 +219542.361}
SPL {X  -165.650, Y  +654.020, Z    +0.000, E1   +29.754, E3 +219542.515}
SPL {X  -165.650, Y  +644.843, Z    +0.000, E1   +43.427, E3 +219540.841}
SPL {X  -165.650, Y  +632.102, Z    +0.000, E1   +56.225, E3 +219540.190}
SPL {X  -165.650, Y  +581.672, Z    +0.000, E1   +69.744, E3 +219552.582}
SPL {X  -165.650, Y  +458.048, Z    +0.000, E1   +68.782, E3 +219633.315}
ENDSPLINE

SPLINE
SPL {X  -165.650, Y  +484.472, Z    +0.000, E1   +63.918, E3 +219647.565}
ENDSPLINE

SPLINE
SPL {X  -165.650, Y  +477.868, Z    +0.000, E1   +63.324, E3 +219658.743}
SPL {X  -165.650, Y  +463.578, Z    +0.000, E1   +63.625, E3 +219671.097}
SPL {X  -165.650, Y  +453.769, Z    +0.000, E1   +63.450, E3 +219682.355}
SPL {X  -165.650, Y  +444.234, Z    +0.000, E1   +63.262, E3 +219693.528}
SPL {X  -165.650, Y  +432.479, Z    +0.000, E1   +63.557, E3 +219703.348}
SPL {X  -165.650, Y  +422.068, Z    +0.000, E1   +63.630, E3 +219713.444}
SPL {X  -165.650, Y  +411.650, Z    +0.000, E1   +63.439, E3 +219725.462}
SPL {X  -165.650, Y  +399.089, Z    +0.000, E1   +63.334, E3 +219739.187}
ENDSPLINE

SPLINE
SPL {X  -165.650, Y  +410.094, Z    +0.000, E1   +60.049, E3 +219749.905}
ENDSPLINE

SPLINE
SPL {X  -165.650, Y  +398.700, Z    +0.000, E1   +60.415, E3 +219760.803}
SPL {X  -165.650, Y  +380.643, Z    +0.000, E1   +61.187, E3 +219776.164}
SPL {X  -165.125, Y  +365.326, Z    +0.000, E1   +61.696, E3 +219789.508}
SPL {X  -164.823, Y  +361.969, Z    +0.000, E1   +60.899, E3 +219798.743}
SPL {X  -163.414, Y  +351.372, Z    +0.000, E1   +61.284, E3 +219808.005}
SPL {X  -162.189, Y  +344.818, Z    +0.000, E1   +60.900, E3 +219817.859}
SPL {X  -160.769, Y  +338.584, Z    +0.000, E1   +60.413, E3 +219828.034}
SPL {X  -157.780, Y  +328.049, Z    +0.000, E1   +60.445, E3 +219839.701}
SPL {X  -155.286, Y  +320.826, Z    +0.000, E1   +59.686, E3 +219852.257}
SPL {X  -152.445, Y  +313.689, Z    +0.000, E1   +59.490, E3 +219861.322}
SPL {X  -149.851, Y  +307.898, Z    +0.000, E1   +58.978, E3 +219870.644}
SPL {X  -146.926, Y  +301.997, Z    +0.000, E1   +58.334, E3 +219880.606}
SPL {X  -143.997, Y  +296.618, Z    +0.000, E1   +58.069, E3 +219887.864}
SPL {X  -142.530, Y  +294.089, Z    +0.000, E1   +57.567, E3 +219893.047}
SPL {X  -134.010, Y  +281.128, Z    +0.000, E1   +60.923, E3 +219891.153}
SPL {X   -93.591, Y  +241.823, Z    +0.000, E1   +55.455, E3 +219983.691}
ENDSPLINE

SPLINE
SPL {X  -110.554, Y  +255.140, Z    +0.000, E1   +52.082, E3 +220110.647}
SPL {X  -137.038, Y  +285.439, Z    +0.000, E1   +46.261, E3 +220130.387}
SPL {X  -149.954, Y  +308.117, Z    +0.000, E1   +39.560, E3 +220136.734}
SPL {X  -160.070, Y  +335.868, Z    +0.000, E1   +27.320, E3 +220131.133}
SPL {X  -163.969, Y  +354.959, Z    +0.000, E1   +17.178, E3 +220131.647}
SPL {X  -165.261, Y  +367.153, Z    +0.000, E1    +9.611, E3 +220130.800}
SPL {X  -165.600, Y  +374.440, Z    +0.000, E1    +4.699, E3 +220130.061}
SPL {X  -165.650, Y  +380.303, Z    +0.000, E1    +0.337, E3 +220129.271}
SPL {X  -165.650, Y  +382.684, Z    +0.000, E1    -2.314, E3 +220128.766}
SPL {X  -165.650, Y  +385.555, Z    +0.000, E1    -6.051, E3 +220127.979}
SPL {X  -165.650, Y  +388.884, Z    +0.000, E1   -10.835, E3 +220128.679}
SPL {X  -165.650, Y  +393.198, Z    +0.000, E1   -17.733, E3 +220127.228}
SPL {X  -165.650, Y  +399.991, Z    +0.000, E1   -27.922, E3 +220128.124}
SPL {X  -165.650, Y  +409.148, Z    +0.000, E1   -43.235, E3 +220123.510}
SPL {X  -165.650, Y  +420.563, Z    +0.000, E1   -54.059, E3 +220124.068}
SPL {X  -165.650, Y  +436.566, Z    +0.000, E1   -62.888, E3 +220125.781}
SPL {X  -165.650, Y  +479.770, Z    +0.000, E1   -67.621, E3 +220145.120}
SPL {X  -165.650, Y  +594.725, Z    +0.000, E1   -69.155, E3 +220212.582}
ENDSPLINE

SPLINE
SPL {X  -165.650, Y  +565.175, Z    +0.000, E1   -62.653, E3 +220236.073}
ENDSPLINE

SPLINE
SPL {X  -165.650, Y  +576.067, Z    +0.000, E1   -62.373, E3 +220249.474}
SPL {X  -165.650, Y  +586.101, Z    +0.000, E1   -62.398, E3 +220260.056}
SPL {X  -165.650, Y  +596.110, Z    +0.000, E1   -62.302, E3 +220271.497}
SPL {X  -165.650, Y  +607.052, Z    +0.000, E1   -62.387, E3 +220282.564}
SPL {X  -165.650, Y  +615.372, Z    +0.000, E1   -62.260, E3 +220292.391}
SPL {X  -165.650, Y  +628.571, Z    +0.000, E1   -62.348, E3 +220306.112}
SPL {X  -165.650, Y  +640.498, Z    +0.000, E1   -62.343, E3 +220318.733}
SPL {X  -165.650, Y  +654.166, Z    +0.000, E1   -62.507, E3 +220332.384}
SPL {X  -165.650, Y  +665.926, Z    +0.000, E1   -62.171, E3 +220347.183}
SPL {X  -165.600, Y  +679.566, Z    +0.000, E1   -62.408, E3 +220360.220}
SPL {X  -165.066, Y  +689.394, Z    +0.000, E1   -62.143, E3 +220372.549}
SPL {X  -164.056, Y  +698.425, Z    +0.000, E1   -62.113, E3 +220382.470}
SPL {X  -162.891, Y  +705.608, Z    +0.000, E1   -61.899, E3 +220391.641}
SPL {X  -160.709, Y  +715.657, Z    +0.000, E1   -61.639, E3 +220404.393}
SPL {X  -157.706, Y  +726.183, Z    +0.000, E1   -61.153, E3 +220418.776}
SPL {X  -155.057, Y  +733.785, Z    +0.000, E1   -60.834, E3 +220428.766}
SPL {X  -152.882, Y  +739.274, Z    +0.000, E1   -60.485, E3 +220436.758}
SPL {X  -150.387, Y  +744.953, Z    +0.000, E1   -60.023, E3 +220445.433}
SPL {X  -146.839, Y  +752.170, Z    +0.000, E1   -59.458, E3 +220456.392}
SPL {X  -142.415, Y  +760.104, Z    +0.000, E1   -58.730, E3 +220468.451}
SPL {X  -132.386, Y  +775.068, Z    +0.000, E1   -61.559, E3 +220470.519}
SPL {X   -89.692, Y  +814.767, Z    +0.000, E1   -54.641, E3 +220584.569}
ENDSPLINE

SPLINE
SPL {X  -133.336, Y  +773.792, Z    +0.000, E1   -47.991, E3 +220713.036}
SPL {X  -153.017, Y  +738.949, Z    +0.000, E1   -37.928, E3 +220726.439}
SPL {X  -160.146, Y  +717.846, Z    +0.000, E1   -27.412, E3 +220713.986}
SPL {X  -163.639, Y  +701.236, Z    +0.000, E1   -18.901, E3 +220720.127}
SPL {X  -165.058, Y  +689.494, Z    +0.000, E1   -11.557, E3 +220718.944}
SPL {X  -165.574, Y  +680.514, Z    +0.000, E1    -5.500, E3 +220718.188}
SPL {X  -165.650, Y  +673.883, Z    +0.000, E1    -0.454, E3 +220717.199}
SPL {X  -165.650, Y  +672.004, Z    +0.000, E1    +1.620, E3 +220716.405}
SPL {X  -165.650, Y  +669.258, Z    +0.000, E1    +5.269, E3 +220716.023}
SPL {X  -165.650, Y  +665.011, Z    +0.000, E1   +11.627, E3 +220715.910}
SPL {X  -165.650, Y  +659.446, Z    +0.000, E1   +21.123, E3 +220714.774}
SPL {X  -165.650, Y  +654.020, Z    +0.000, E1   +29.754, E3 +220714.929}
SPL {X  -165.650, Y  +644.843, Z    +0.000, E1   +43.427, E3 +220713.255}
SPL {X  -165.650, Y  +632.102, Z    +0.000, E1   +56.225, E3 +220712.604}
SPL {X  -165.650, Y  +581.672, Z    +0.000, E1   +69.744, E3 +220724.996}
SPL {X  -165.650, Y  +458.048, Z    +0.000, E1   +68.782, E3 +220805.728}
ENDSPLINE

SPLINE
SPL {X  -165.650, Y  +484.472, Z    +0.000, E1   +63.918, E3 +220819.979}
ENDSPLINE

SPLINE
SPL {X  -165.650, Y  +477.868, Z    +0.000, E1   +63.324, E3 +220831.157}
SPL {X  -165.650, Y  +463.578, Z    +0.000, E1   +63.625, E3 +220843.511}
SPL {X  -165.650, Y  +453.769, Z    +0.000, E1   +63.450, E3 +220854.769}
SPL {X  -165.650, Y  +444.234, Z    +0.000, E1   +63.262, E3 +220865.942}
SPL {X  -165.650, Y  +432.479, Z    +0.000, E1   +63.557, E3 +220875.762}
SPL {X  -165.650, Y  +422.068, Z    +0.000, E1   +63.630, E3 +220885.857}
SPL {X  -165.650, Y  +411.650, Z    +0.000, E1   +63.439, E3 +220897.876}
SPL {X  -165.650, Y  +399.089, Z    +0.000, E1   +63.334, E3 +220911.601}
ENDSPLINE

SPLINE
SPL {X  -165.650, Y  +410.094, Z    +0.000, E1   +60.049, E3 +220922.319}
ENDSPLINE

SPLINE
SPL {X  -165.650, Y  +398.700, Z    +0.000, E1   +60.415, E3 +220933.216}
SPL {X  -165.650, Y  +380.643, Z    +0.000, E1   +61.187, E3 +220948.578}
SPL {X  -165.125, Y  +365.326, Z    +0.000, E1   +61.696, E3 +220961.922}
SPL {X  -164.823, Y  +361.969, Z    +0.000, E1   +60.899, E3 +220971.157}
SPL {X  -163.414, Y  +351.372, Z    +0.000, E1   +61.284, E3 +220980.419}
SPL {X  -162.189, Y  +344.818, Z    +0.000, E1   +60.900, E3 +220990.272}
SPL {X  -160.769, Y  +338.584, Z    +0.000, E1   +60.413, E3 +221000.448}
SPL {X  -157.780, Y  +328.049, Z    +0.000, E1   +60.445, E3 +221012.115}
SPL {X  -155.286, Y  +320.826, Z    +0.000, E1   +59.686, E3 +221024.671}
SPL {X  -152.445, Y  +313.689, Z    +0.000, E1   +59.490, E3 +221033.736}
SPL {X  -150.678, Y  +309.680, Z    +0.000, E1   +58.971, E3 +221041.048}
SPL {X  -148.010, Y  +304.117, Z    +0.000, E1   +58.696, E3 +221048.795}
SPL {X  -144.822, Y  +298.086, Z    +0.000, E1   +58.093, E3 +221058.577}
SPL {X  -142.530, Y  +294.089, Z    +0.000, E1   +57.567, E3 +221065.461}
SPL {X  -134.010, Y  +281.128, Z    +0.000, E1   +60.923, E3 +221063.567}
SPL {X   -93.591, Y  +241.823, Z    +0.000, E1   +55.455, E3 +221156.105}
ENDSPLINE

SPLINE
SPL {X  -110.554, Y  +255.140, Z    +0.000, E1   +52.082, E3 +221283.061}
SPL {X  -144.988, Y  +298.385, Z    +0.000, E1   +42.755, E3 +221306.880}
SPL {X  -160.070, Y  +335.868, Z    +0.000, E1   +27.320, E3 +221303.547}
SPL {X  -163.969, Y  +354.959, Z    +0.000, E1   +17.178, E3 +221304.061}
SPL {X  -165.261, Y  +367.153, Z    +0.000, E1    +9.611, E3 +221303.213}
SPL {X  -165.600, Y  +374.440, Z    +0.000, E1    +4.699, E3 +221302.474}
SPL {X  -165.650, Y  +380.303, Z    +0.000, E1    +0.337, E3 +221301.685}
SPL {X  -165.650, Y  +382.684, Z    +0.000, E1    -2.314, E3 +221301.179}
SPL {X  -165.650, Y  +386.855, Z    +0.000, E1    -7.700, E3 +221300.666}
SPL {X  -165.650, Y  +393.198, Z    +0.000, E1   -17.733, E3 +221299.642}
SPL {X  -165.650, Y  +399.991, Z    +0.000, E1   -27.922, E3 +221300.538}
SPL {X  -165.650, Y  +409.148, Z    +0.000, E1   -43.235, E3 +221295.924}
SPL {X  -165.650, Y  +420.563, Z    +0.000, E1   -54.059, E3 +221296.482}
SPL {X  -165.650, Y  +436.566, Z    +0.000, E1   -62.888, E3 +221298.195}
SPL {X  -165.650, Y  +479.770, Z    +0.000, E1   -67.621, E3 +221317.534}
SPL {X  -165.650, Y  +594.725, Z    +0.000, E1   -69.155, E3 +221384.996}
ENDSPLINE

SPLINE
SPL {X  -165.650, Y  +565.175, Z    +0.000, E1   -62.653, E3 +221408.486}
ENDSPLINE

SPLINE
SPL {X  -165.650, Y  +576.067, Z    +0.000, E1   -62.373, E3 +221421.888}
SPL {X  -165.650, Y  +586.101, Z    +0.000, E1   -62.398, E3 +221432.470}
SPL {X  -165.650, Y  +596.110, Z    +0.000, E1   -62.302, E3 +221443.910}
SPL {X  -165.650, Y  +607.052, Z    +0.000, E1   -62.387, E3 +221454.978}
SPL {X  -165.650, Y  +618.920, Z    +0.000, E1   -62.340, E3 +221468.168}
SPL {X  -165.650, Y  +635.445, Z    +0.000, E1   -62.341, E3 +221485.969}
SPL {X  -165.650, Y  +654.166, Z    +0.000, E1   -62.507, E3 +221504.798}
SPL {X  -165.650, Y  +665.926, Z    +0.000, E1   -62.171, E3 +221519.597}
SPL {X  -165.644, Y  +676.899, Z    +0.000, E1   -62.447, E3 +221529.364}
SPL {X  -165.241, Y  +687.133, Z    +0.000, E1   -62.230, E3 +221542.066}
SPL {X  -164.056, Y  +698.425, Z    +0.000, E1   -62.113, E3 +221554.883}
SPL {X  -162.891, Y  +705.608, Z    +0.000, E1   -61.899, E3 +221564.055}
SPL {X  -160.709, Y  +715.657, Z    +0.000, E1   -61.639, E3 +221576.807}
SPL {X  -157.706, Y  +726.183, Z    +0.000, E1   -61.153, E3 +221591.190}
SPL {X  -155.057, Y  +733.785, Z    +0.000, E1   -60.834, E3 +221601.179}
SPL {X  -152.882, Y  +739.274, Z    +0.000, E1   -60.485, E3 +221609.172}
SPL {X  -150.387, Y  +744.953, Z    +0.000, E1   -60.023, E3 +221617.847}
SPL {X  -147.728, Y  +750.443, Z    +0.000, E1   -59.568, E3 +221626.231}
SPL {X  -143.895, Y  +757.561, Z    +0.000, E1   -58.980, E3 +221636.967}
SPL {X  -141.017, Y  +762.414, Z    +0.000, E1   -58.435, E3 +221644.548}
SPL {X  -134.606, Y  +772.046, Z    +0.000, E1   -61.105, E3 +221642.194}
SPL {X  -127.075, Y  +781.763, Z    +0.000, E1   -62.555, E3 +221644.508}
SPL {X   -89.692, Y  +814.767, Z    +0.000, E1   -54.641, E3 +221756.982}
ENDSPLINE

SPLINE
SPL {X  -133.336, Y  +773.792, Z    +0.000, E1   -47.991, E3 +221885.449}
SPL {X  -153.017, Y  +738.949, Z    +0.000, E1   -37.928, E3 +221898.853}
SPL {X  -160.146, Y  +717.846, Z    +0.000, E1   -27.412, E3 +221886.400}
SPL {X  -163.639, Y  +701.236, Z    +0.000, E1   -18.901, E3 +221892.541}
SPL {X  -165.380, Y  +684.951, Z    +0.000, E1    -8.606, E3 +221890.798}
SPL {X  -165.650, Y  +675.640, Z    +0.000, E1    -1.874, E3 +221890.334}
SPL {X  -165.650, Y  +672.727, Z    +0.000, E1    +0.658, E3 +221889.084}
SPL {X  -165.650, Y  +669.258, Z    +0.000, E1    +5.269, E3 +221888.437}
SPL {X  -165.650, Y  +665.011, Z    +0.000, E1   +11.627, E3 +221888.324}
SPL {X  -165.650, Y  +659.446, Z    +0.000, E1   +21.123, E3 +221887.188}
SPL {X  -165.650, Y  +654.020, Z    +0.000, E1   +29.754, E3 +221887.343}
SPL {X  -165.650, Y  +644.843, Z    +0.000, E1   +43.427, E3 +221885.669}
SPL {X  -165.650, Y  +632.102, Z    +0.000, E1   +56.225, E3 +221885.017}
SPL {X  -165.650, Y  +581.672, Z    +0.000, E1   +69.744, E3 +221897.410}
SPL {X  -165.650, Y  +455.882, Z    +0.000, E1   +70.075, E3 +221969.674}
ENDSPLINE

SPLINE
SPL {X  -165.650, Y  +480.501, Z    +0.000, E1   +64.561, E3 +221991.643}
ENDSPLINE

SPLINE
SPL {X  -165.650, Y  +477.868, Z    +0.000, E1   +63.324, E3 +222003.571}
SPL {X  -165.650, Y  +463.578, Z    +0.000, E1   +63.625, E3 +222015.924}
SPL {X  -165.650, Y  +453.769, Z    +0.000, E1   +63.450, E3 +222027.183}
SPL {X  -165.650, Y  +444.234, Z    +0.000, E1   +63.262, E3 +222038.356}
SPL {X  -165.650, Y  +432.479, Z    +0.000, E1   +63.557, E3 +222048.176}
SPL {X  -165.650, Y  +422.068, Z    +0.000, E1   +63.630, E3 +222058.271}
SPL {X  -165.650, Y  +409.231, Z    +0.000, E1   +63.364, E3 +222073.520}
SPL {X  -165.650, Y  +395.008, Z    +0.000, E1   +63.445, E3 +222087.283}
ENDSPLINE

SPLINE
SPL {X  -165.650, Y  +410.094, Z    +0.000, E1   +60.049, E3 +222094.732}
ENDSPLINE

SPLINE
SPL {X  -165.650, Y  +398.700, Z    +0.000, E1   +60.415, E3 +222105.630}
SPL {X  -165.650, Y  +380.643, Z    +0.000, E1   +61.187, E3 +222120.992}
SPL {X  -165.125, Y  +365.326, Z    +0.000, E1   +61.696, E3 +222134.335}
SPL {X  -164.823, Y  +361.969, Z    +0.000, E1   +60.899, E3 +222143.570}
SPL {X  -163.414, Y  +351.372, Z    +0.000, E1   +61.284, E3 +222152.833}
SPL {X  -162.189, Y  +344.818, Z    +0.000, E1   +60.900, E3 +222162.686}
SPL {X  -160.769, Y  +338.584, Z    +0.000, E1   +60.413, E3 +222172.862}
SPL {X  -157.780, Y  +328.049, Z    +0.000, E1   +60.445, E3 +222184.529}
SPL {X  -155.286, Y  +320.826, Z    +0.000, E1   +59.686, E3 +222197.084}
SPL {X  -152.445, Y  +313.689, Z    +0.000, E1   +59.490, E3 +222206.150}
SPL {X  -149.851, Y  +307.898, Z    +0.000, E1   +58.978, E3 +222215.472}
SPL {X  -146.926, Y  +301.997, Z    +0.000, E1   +58.334, E3 +222225.433}
SPL {X  -143.281, Y  +295.370, Z    +0.000, E1   +57.860, E3 +222235.202}
SPL {X  -134.010, Y  +281.128, Z    +0.000, E1   +60.923, E3 +222235.980}
SPL {X   -93.591, Y  +241.823, Z    +0.000, E1   +55.455, E3 +222328.518}
ENDSPLINE

SPLINE
SPL {X  -110.554, Y  +255.140, Z    +0.000, E1   +52.082, E3 +222455.474}
SPL {X  -137.038, Y  +285.439, Z    +0.000, E1   +46.261, E3 +222475.214}
SPL {X  -149.954, Y  +308.117, Z    +0.000, E1   +39.560, E3 +222481.562}
SPL {X  -160.070, Y  +335.868, Z    +0.000, E1   +27.320, E3 +222475.960}
SPL {X  -163.969, Y  +354.959, Z    +0.000, E1   +17.178, E3 +222476.475}
SPL {X  -165.261, Y  +367.153, Z    +0.000, E1    +9.611, E3 +222475.627}
SPL {X  -165.600, Y  +374.440, Z    +0.000, E1    +4.699, E3 +222474.888}
SPL {X  -165.650, Y  +379.657, Z    +0.000, E1    +0.819, E3 +222474.417}
SPL {X  -165.650, Y  +381.885, Z    +0.000, E1    -1.282, E3 +222473.661}
SPL {X  -165.650, Y  +386.855, Z    +0.000, E1    -7.700, E3 +222473.080}
SPL {X  -165.650, Y  +393.198, Z    +0.000, E1   -17.733, E3 +222472.056}
SPL {X  -165.650, Y  +399.991, Z    +0.000, E1   -27.922, E3 +222472.952}
SPL {X  -165.650, Y  +409.148, Z    +0.000, E1   -43.235, E3 +222468.338}
SPL {X  -165.650, Y  +420.563, Z    +0.000, E1   -54.059, E3 +222468.896}
SPL {X  -165.650, Y  +436.566, Z    +0.000, E1   -62.888, E3 +222470.609}
SPL {X  -165.650, Y  +479.770, Z    +0.000, E1   -67.621, E3 +222489.947}
SPL {X  -165.650, Y  +594.725, Z    +0.000, E1   -69.155, E3 +222557.409}
ENDSPLINE

SPLINE
SPL {X  -165.650, Y  +565.175, Z    +0.000, E1   -62.653, E3 +222580.900}
ENDSPLINE

SPLINE
SPL {X  -165.650, Y  +576.067, Z    +0.000, E1   -62.373, E3 +222594.301}
SPL {X  -165.650, Y  +586.101, Z    +0.000, E1   -62.398, E3 +222604.883}
SPL {X  -165.650, Y  +596.110, Z    +0.000, E1   -62.302, E3 +222616.324}
SPL {X  -165.650, Y  +607.052, Z    +0.000, E1   -62.387, E3 +222627.391}
SPL {X  -165.650, Y  +618.920, Z    +0.000, E1   -62.340, E3 +222640.582}
SPL {X  -165.650, Y  +631.247, Z    +0.000, E1   -62.270, E3 +222654.198}
SPL {X  -165.650, Y  +645.288, Z    +0.000, E1   -62.475, E3 +222667.878}
SPL {X  -165.650, Y  +657.265, Z    +0.000, E1   -62.410, E3 +222680.997}
SPL {X  -165.650, Y  +665.926, Z    +0.000, E1   -62.171, E3 +222692.010}
SPL {X  -165.644, Y  +676.899, Z    +0.000, E1   -62.447, E3 +222701.778}
SPL {X  -165.241, Y  +687.133, Z    +0.000, E1   -62.230, E3 +222714.480}
SPL {X  -164.056, Y  +698.425, Z    +0.000, E1   -62.113, E3 +222727.297}
SPL {X  -162.891, Y  +705.608, Z    +0.000, E1   -61.899, E3 +222736.469}
SPL {X  -160.709, Y  +715.657, Z    +0.000, E1   -61.639, E3 +222749.221}
SPL {X  -157.706, Y  +726.183, Z    +0.000, E1   -61.153, E3 +222763.603}
SPL {X  -155.057, Y  +733.785, Z    +0.000, E1   -60.834, E3 +222773.593}
SPL {X  -152.882, Y  +739.274, Z    +0.000, E1   -60.485, E3 +222781.586}
SPL {X  -150.387, Y  +744.953, Z    +0.000, E1   -60.023, E3 +222790.261}
SPL {X  -146.839, Y  +752.170, Z    +0.000, E1   -59.458, E3 +222801.220}
SPL {X  -142.415, Y  +760.104, Z    +0.000, E1   -58.730, E3 +222813.278}
SPL {X  -132.386, Y  +775.068, Z    +0.000, E1   -61.559, E3 +222815.347}
SPL {X   -89.692, Y  +814.767, Z    +0.000, E1   -54.641, E3 +222929.396}
ENDSPLINE

SPLINE
SPL {X  -120.253, Y  +789.426, Z    +0.000, E1   -51.165, E3 +223050.670}
SPL {X  -143.101, Y  +758.939, Z    +0.000, E1   -44.365, E3 +223064.778}
SPL {X  -158.740, Y  +722.846, Z    +0.000, E1   -30.140, E3 +223062.817}
SPL {X  -163.639, Y  +701.236, Z    +0.000, E1   -18.901, E3 +223064.955}
SPL {X  -165.058, Y  +689.494, Z    +0.000, E1   -11.557, E3 +223063.772}
SPL {X  -165.574, Y  +680.514, Z    +0.000, E1    -5.500, E3 +223063.015}
SPL {X  -165.650, Y  +673.883, Z    +0.000, E1    -0.454, E3 +223062.026}
SPL {X  -165.650, Y  +672.004, Z    +0.000, E1    +1.620, E3 +223061.232}
SPL {X  -165.650, Y  +669.258, Z    +0.000, E1    +5.269, E3 +223060.851}
SPL {X  -165.650, Y  +665.011, Z    +0.000, E1   +11.627, E3 +223060.738}
SPL {X  -165.650, Y  +659.446, Z    +0.000, E1   +21.123, E3 +223059.602}
SPL {X  -165.650, Y  +654.020, Z    +0.000, E1   +29.754, E3 +223059.756}
SPL {X  -165.650, Y  +644.843, Z    +0.000, E1   +43.427, E3 +223058.082}
SPL {X  -165.650, Y  +632.102, Z    +0.000, E1   +56.225, E3 +223057.431}
SPL {X  -165.650, Y  +581.672, Z    +0.000, E1   +69.744, E3 +223069.823}
SPL {X  -165.650, Y  +458.048, Z    +0.000, E1   +68.782, E3 +223150.556}
ENDSPLINE

SPLINE
SPL {X  -165.650, Y  +484.472, Z    +0.000, E1   +63.918, E3 +223164.807}
ENDSPLINE

SPLINE
SPL {X  -165.650, Y  +477.868, Z    +0.000, E1   +63.324, E3 +223175.984}
SPL {X  -165.650, Y  +463.578, Z    +0.000, E1   +63.625, E3 +223188.338}
SPL {X  -165.650, Y  +453.769, Z    +0.000, E1   +63.450, E3 +223199.597}
SPL {X  -165.650, Y  +444.234, Z    +0.000, E1   +63.262, E3 +223210.770}
SPL {X  -165.650, Y  +432.479, Z    +0.000, E1   +63.557, E3 +223220.590}
SPL {X  -165.650, Y  +422.068, Z    +0.000, E1   +63.630, E3 +223230.685}
SPL {X  -165.650, Y  +411.650, Z    +0.000, E1   +63.439, E3 +223242.703}
SPL {X  -165.650, Y  +399.089, Z    +0.000, E1   +63.334, E3 +223256.429}
ENDSPLINE

SPLINE
SPL {X  -165.650, Y  +410.094, Z    +0.000, E1   +60.049, E3 +223267.146}
ENDSPLINE

SPLINE
SPL {X  -165.650, Y  +398.700, Z    +0.000, E1   +60.415, E3 +223278.044}
SPL {X  -165.650, Y  +380.643, Z    +0.000, E1   +61.187, E3 +223293.406}
SPL {X  -165.125, Y  +365.326, Z    +0.000, E1   +61.696, E3 +223306.749}
SPL {X  -164.823, Y  +361.969, Z    +0.000, E1   +60.899, E3 +223315.984}
SPL {X  -163.414, Y  +351.372, Z    +0.000, E1   +61.284, E3 +223325.247}
SPL {X  -162.189, Y  +344.818, Z    +0.000, E1   +60.900, E3 +223335.100}
SPL {X  -160.769, Y  +338.584, Z    +0.000, E1   +60.413, E3 +223345.276}
SPL {X  -157.780, Y  +328.049, Z    +0.000, E1   +60.445, E3 +223356.943}
SPL {X  -155.286, Y  +320.826, Z    +0.000, E1   +59.686, E3 +223369.498}
SPL {X  -152.445, Y  +313.689, Z    +0.000, E1   +59.490, E3 +223378.564}
SPL {X  -149.851, Y  +307.898, Z    +0.000, E1   +58.978, E3 +223387.886}
SPL {X  -146.926, Y  +301.997, Z    +0.000, E1   +58.334, E3 +223397.847}
SPL {X  -143.997, Y  +296.618, Z    +0.000, E1   +58.069, E3 +223405.105}
SPL {X  -142.530, Y  +294.089, Z    +0.000, E1   +57.567, E3 +223410.289}
SPL {X  -134.010, Y  +281.128, Z    +0.000, E1   +60.923, E3 +223408.394}
SPL {X   -93.591, Y  +241.823, Z    +0.000, E1   +55.455, E3 +223500.932}
ENDSPLINE

SPLINE
SPL {X  -110.554, Y  +255.140, Z    +0.000, E1   +52.082, E3 +223627.888}
SPL {X  -137.038, Y  +285.439, Z    +0.000, E1   +46.261, E3 +223647.628}
SPL {X  -149.954, Y  +308.117, Z    +0.000, E1   +39.560, E3 +223653.976}
SPL {X  -160.070, Y  +335.868, Z    +0.000, E1   +27.320, E3 +223648.374}
SPL {X  -163.969, Y  +354.959, Z    +0.000, E1   +17.178, E3 +223648.888}
SPL {X  -165.261, Y  +367.153, Z    +0.000, E1    +9.611, E3 +223648.041}
SPL {X  -165.600, Y  +374.440, Z    +0.000, E1    +4.699, E3 +223647.302}
SPL {X  -165.650, Y  +380.303, Z    +0.000, E1    +0.337, E3 +223646.513}
SPL {X  -165.650, Y  +382.684, Z    +0.000, E1    -2.314, E3 +223646.007}
SPL {X  -165.650, Y  +385.555, Z    +0.000, E1    -6.051, E3 +223645.220}
SPL {X  -165.650, Y  +388.884, Z    +0.000, E1   -10.835, E3 +223645.920}
SPL {X  -165.650, Y  +393.198, Z    +0.000, E1   -17.733, E3 +223644.470}
SPL {X  -165.650, Y  +399.991, Z    +0.000, E1   -27.922, E3 +223645.365}
SPL {X  -165.650, Y  +409.148, Z    +0.000, E1   -43.235, E3 +223640.752}
SPL {X  -165.650, Y  +420.563, Z    +0.000, E1   -54.059, E3 +223641.310}
SPL {X  -165.650, Y  +436.566, Z    +0.000, E1   -62.888, E3 +223643.022}
SPL {X  -165.650, Y  +479.770, Z    +0.000, E1   -67.621, E3 +223662.361}
SPL {X  -165.650, Y  +594.725, Z    +0.000, E1   -69.155, E3 +223729.823}
ENDSPLINE

SPLINE
SPL {X  -165.650, Y  +562.482, Z    +0.000, E1   -62.785, E3 +223749.289}
ENDSPLINE

SPLINE
SPL {X  -165.650, Y  +572.898, Z    +0.000, E1   -62.409, E3 +223763.226}
SPL {X  -165.650, Y  +586.101, Z    +0.000, E1   -62.398, E3 +223777.297}
SPL {X  -165.650, Y  +596.110, Z    +0.000, E1   -62.302, E3 +223788.738}
SPL {X  -165.650, Y  +607.052, Z    +0.000, E1   -62.387, E3 +223799.805}
SPL {X  -165.650, Y  +615.372, Z    +0.000, E1   -62.260, E3 +223809.632}
SPL {X  -165.650, Y  +628.571, Z    +0.000, E1   -62.348, E3 +223823.353}
SPL {X  -165.650, Y  +640.498, Z    +0.000, E1   -62.343, E3 +223835.974}
SPL {X  -165.650, Y  +654.166, Z    +0.000, E1   -62.507, E3 +223849.626}
SPL {X  -165.650, Y  +665.926, Z    +0.000, E1   -62.171, E3 +223864.424}
SPL {X  -165.600, Y  +679.566, Z    +0.000, E1   -62.408, E3 +223877.461}
SPL {X  -165.066, Y  +689.394, Z    +0.000, E1   -62.143, E3 +223889.791}
SPL {X  -164.056, Y  +698.425, Z    +0.000, E1   -62.113, E3 +223899.711}
SPL {X  -162.891, Y  +705.608, Z    +0.000, E1   -61.899, E3 +223908.882}
SPL {X  -161.308, Y  +713.180, Z    +0.000, E1   -61.813, E3 +223917.576}
SPL {X  -160.182, Y  +717.709, Z    +0.000, E1   -61.401, E3 +223925.188}
SPL {X  -157.706, Y  +726.183, Z    +0.000, E1   -61.153, E3 +223936.017}
SPL {X  -155.057, Y  +733.785, Z    +0.000, E1   -60.834, E3 +223946.007}
SPL {X  -152.882, Y  +739.274, Z    +0.000, E1   -60.485, E3 +223954.000}
SPL {X  -149.755, Y  +746.304, Z    +0.000, E1   -59.867, E3 +223965.121}
SPL {X  -146.068, Y  +753.629, Z    +0.000, E1   -59.384, E3 +223975.480}
SPL {X  -143.119, Y  +758.908, Z    +0.000, E1   -58.828, E3 +223983.855}
SPL {X  -141.017, Y  +762.414, Z    +0.000, E1   -58.435, E3 +223989.375}
SPL {X  -132.386, Y  +775.068, Z    +0.000, E1   -61.559, E3 +223987.761}
SPL {X   -89.692, Y  +814.767, Z    +0.000, E1   -54.641, E3 +224101.810}
ENDSPLINE

SPLINE
SPL {X  -133.336, Y  +773.792, Z    +0.000, E1   -47.991, E3 +224230.277}
SPL {X  -153.017, Y  +738.949, Z    +0.000, E1   -37.928, E3 +224243.681}
SPL {X  -160.146, Y  +717.846, Z    +0.000, E1   -27.412, E3 +224231.227}
SPL {X  -163.639, Y  +701.236, Z    +0.000, E1   -18.901, E3 +224237.368}
SPL {X  -165.058, Y  +689.494, Z    +0.000, E1   -11.557, E3 +224236.185}
SPL {X  -165.574, Y  +680.514, Z    +0.000, E1    -5.500, E3 +224235.429}
SPL {X  -165.650, Y  +673.883, Z    +0.000, E1    -0.454, E3 +224234.440}
SPL {X  -165.650, Y  +672.004, Z    +0.000, E1    +1.620, E3 +224233.646}
SPL {X  -165.650, Y  +669.258, Z    +0.000, E1    +5.269, E3 +224233.264}
SPL {X  -165.650, Y  +665.011, Z    +0.000, E1   +11.627, E3 +224233.152}
SPL {X  -165.650, Y  +659.446, Z    +0.000, E1   +21.123, E3 +224232.016}
SPL {X  -165.650, Y  +654.020, Z    +0.000, E1   +29.754, E3 +224232.170}
SPL {X  -165.650, Y  +644.843, Z    +0.000, E1   +43.427, E3 +224230.496}
SPL {X  -165.650, Y  +632.102, Z    +0.000, E1   +56.225, E3 +224229.845}
SPL {X  -165.650, Y  +581.672, Z    +0.000, E1   +69.744, E3 +224242.237}
SPL {X  -165.650, Y  +458.048, Z    +0.000, E1   +68.782, E3 +224322.970}
ENDSPLINE

SPLINE
SPL {X  -165.650, Y  +484.472, Z    +0.000, E1   +63.918, E3 +224337.221}
ENDSPLINE

SPLINE
SPL {X  -165.650, Y  +477.868, Z    +0.000, E1   +63.324, E3 +224348.398}
SPL {X  -165.650, Y  +463.578, Z    +0.000, E1   +63.625, E3 +224360.752}
SPL {X  -165.650, Y  +453.769, Z    +0.000, E1   +63.450, E3 +224372.011}
SPL {X  -165.650, Y  +444.234, Z    +0.000, E1   +63.262, E3 +224383.183}
SPL {X  -165.650, Y  +432.479, Z    +0.000, E1   +63.557, E3 +224393.003}
SPL {X  -165.650, Y  +422.068, Z    +0.000, E1   +63.630, E3 +224403.099}
SPL {X  -165.650, Y  +411.650, Z    +0.000, E1   +63.439, E3 +224415.117}
SPL {X  -165.650, Y  +399.089, Z    +0.000, E1   +63.334, E3 +224428.843}
ENDSPLINE

SPLINE
SPL {X  -165.650, Y  +410.094, Z    +0.000, E1   +60.049, E3 +224439.560}
ENDSPLINE

SPLINE
SPL {X  -165.650, Y  +398.700, Z    +0.000, E1   +60.415, E3 +224450.458}
SPL {X  -165.650, Y  +382.616, Z    +0.000, E1   +61.427, E3 +224461.676}
SPL {X  -165.650, Y  +379.013, Z    +0.000, E1   +60.888, E3 +224469.499}
SPL {X  -165.125, Y  +365.326, Z    +0.000, E1   +61.696, E3 +224479.163}
SPL {X  -164.823, Y  +361.969, Z    +0.000, E1   +60.899, E3 +224488.398}
SPL {X  -163.414, Y  +351.372, Z    +0.000, E1   +61.284, E3 +224497.660}
SPL {X  -162.189, Y  +344.818, Z    +0.000, E1   +60.900, E3 +224507.514}
SPL {X  -160.769, Y  +338.584, Z    +0.000, E1   +60.413, E3 +224517.690}
SPL {X  -157.780, Y  +328.049, Z    +0.000, E1   +60.445, E3 +224529.356}
SPL {X  -155.286, Y  +320.826, Z    +0.000, E1   +59.686, E3 +224541.912}
SPL {X  -151.657, Y  +311.865, Z    +0.000, E1   +59.311, E3 +224554.214}
SPL {X  -147.428, Y  +302.969, Z    +0.000, E1   +58.548, E3 +224568.230}
SPL {X  -143.281, Y  +295.370, Z    +0.000, E1   +57.860, E3 +224580.029}
SPL {X  -134.010, Y  +281.128, Z    +0.000, E1   +60.923, E3 +224580.808}
SPL {X   -93.591, Y  +241.823, Z    +0.000, E1   +55.455, E3 +224673.346}
ENDSPLINE

SPLINE
SPL {X  -110.554, Y  +255.140, Z    +0.000, E1   +52.082, E3 +224800.302}
SPL {X  -137.038, Y  +285.439, Z    +0.000, E1   +46.261, E3 +224820.042}
SPL {X  -149.954, Y  +308.117, Z    +0.000, E1   +39.560, E3 +224826.389}
SPL {X  -160.070, Y  +335.868, Z    +0.000, E1   +27.320, E3 +224820.788}
SPL {X  -163.969, Y  +354.959, Z    +0.000, E1   +17.178, E3 +224821.302}
SPL {X  -165.261, Y  +367.153, Z    +0.000, E1    +9.611, E3 +224820.455}
SPL {X  -165.600, Y  +374.440, Z    +0.000, E1    +4.699, E3 +224819.716}
SPL {X  -165.650, Y  +379.657, Z    +0.000, E1    +0.819, E3 +224819.244}
SPL {X  -165.650, Y  +381.885, Z    +0.000, E1    -1.282, E3 +224818.488}
SPL {X  -165.650, Y  +386.855, Z    +0.000, E1    -7.700, E3 +224817.907}
SPL {X  -165.650, Y  +393.198, Z    +0.000, E1   -17.733, E3 +224816.883}
SPL {X  -165.650, Y  +399.991, Z    +0.000, E1   -27.922, E3 +224817.779}
SPL {X  -165.650, Y  +411.457, Z    +0.000, E1   -45.557, E3 +224813.527}
SPL {X  -165.650, Y  +427.627, Z    +0.000, E1   -58.747, E3 +224814.161}
SPL {X  -165.650, Y  +479.770, Z    +0.000, E1   -67.621, E3 +224834.775}
SPL {X  -165.650, Y  +594.725, Z    +0.000, E1   -69.155, E3 +224902.237}
ENDSPLINE

SPLINE
SPL {X  -165.650, Y  +565.175, Z    +0.000, E1   -62.653, E3 +224925.728}
ENDSPLINE

SPLINE
SPL {X  -165.650, Y  +576.067, Z    +0.000, E1   -62.373, E3 +224939.129}
SPL {X  -165.650, Y  +586.101, Z    +0.000, E1   -62.398, E3 +224949.711}
SPL {X  -165.650, Y  +596.110, Z    +0.000, E1   -62.302, E3 +224961.152}
SPL {X  -165.650, Y  +607.052, Z    +0.000, E1   -62.387, E3 +224972.219}
SPL {X  -165.650, Y  +618.920, Z    +0.000, E1   -62.340, E3 +224985.409}
SPL {X  -165.650, Y  +631.247, Z    +0.000, E1   -62.270, E3 +224999.026}
SPL {X  -165.650, Y  +645.288, Z    +0.000, E1   -62.475, E3 +225012.706}
SPL {X  -165.650, Y  +657.265, Z    +0.000, E1   -62.410, E3 +225025.824}
SPL {X  -165.650, Y  +665.926, Z    +0.000, E1   -62.171, E3 +225036.838}
SPL {X  -165.600, Y  +679.566, Z    +0.000, E1   -62.408, E3 +225049.875}
SPL {X  -165.066, Y  +689.394, Z    +0.000, E1   -62.143, E3 +225062.205}
SPL {X  -164.056, Y  +698.425, Z    +0.000, E1   -62.113, E3 +225072.125}
SPL {X  -162.891, Y  +705.608, Z    +0.000, E1   -61.899, E3 +225081.296}
SPL {X  -161.308, Y  +713.180, Z    +0.000, E1   -61.813, E3 +225089.990}
SPL {X  -160.182, Y  +717.709, Z    +0.000, E1   -61.401, E3 +225097.602}
SPL {X  -157.706, Y  +726.183, Z    +0.000, E1   -61.153, E3 +225108.431}
SPL {X  -155.057, Y  +733.785, Z    +0.000, E1   -60.834, E3 +225118.421}
SPL {X  -152.882, Y  +739.274, Z    +0.000, E1   -60.485, E3 +225126.413}
SPL {X  -150.387, Y  +744.953, Z    +0.000, E1   -60.023, E3 +225135.088}
SPL {X  -147.728, Y  +750.443, Z    +0.000, E1   -59.568, E3 +225143.472}
SPL {X  -143.895, Y  +757.561, Z    +0.000, E1   -58.980, E3 +225154.209}
SPL {X  -141.017, Y  +762.414, Z    +0.000, E1   -58.435, E3 +225161.789}
SPL {X  -134.606, Y  +772.046, Z    +0.000, E1   -61.105, E3 +225159.435}
SPL {X  -127.075, Y  +781.763, Z    +0.000, E1   -62.555, E3 +225161.750}
SPL {X   -89.692, Y  +814.767, Z    +0.000, E1   -54.641, E3 +225274.224}
ENDSPLINE

SPLINE
SPL {X  -133.336, Y  +773.792, Z    +0.000, E1   -47.991, E3 +225402.691}
SPL {X  -153.017, Y  +738.949, Z    +0.000, E1   -37.928, E3 +225416.095}
SPL {X  -160.146, Y  +717.846, Z    +0.000, E1   -27.412, E3 +225403.641}
SPL {X  -163.639, Y  +701.236, Z    +0.000, E1   -18.901, E3 +225409.782}
SPL {X  -165.380, Y  +684.951, Z    +0.000, E1    -8.606, E3 +225408.039}
SPL {X  -165.650, Y  +675.640, Z    +0.000, E1    -1.874, E3 +225407.575}
SPL {X  -165.650, Y  +672.727, Z    +0.000, E1    +0.658, E3 +225406.325}
SPL {X  -165.650, Y  +669.258, Z    +0.000, E1    +5.269, E3 +225405.678}
SPL {X  -165.650, Y  +665.011, Z    +0.000, E1   +11.627, E3 +225405.565}
SPL {X  -165.650, Y  +659.446, Z    +0.000, E1   +21.123, E3 +225404.429}
SPL {X  -165.650, Y  +654.020, Z    +0.000, E1   +29.754, E3 +225404.584}
SPL {X  -165.650, Y  +644.843, Z    +0.000, E1   +43.427, E3 +225402.910}
SPL {X  -165.650, Y  +632.102, Z    +0.000, E1   +56.225, E3 +225402.259}
SPL {X  -165.650, Y  +581.672, Z    +0.000, E1   +69.744, E3 +225414.651}
SPL {X  -165.650, Y  +455.882, Z    +0.000, E1   +70.075, E3 +225486.915}
ENDSPLINE

SPLINE
SPL {X  -165.650, Y  +480.501, Z    +0.000, E1   +64.561, E3 +225508.884}
ENDSPLINE

SPLINE
SPL {X  -165.650, Y  +477.868, Z    +0.000, E1   +63.324, E3 +225520.812}
SPL {X  -165.650, Y  +463.578, Z    +0.000, E1   +63.625, E3 +225533.166}
SPL {X  -165.650, Y  +453.769, Z    +0.000, E1   +63.450, E3 +225544.424}
SPL {X  -165.650, Y  +444.234, Z    +0.000, E1   +63.262, E3 +225555.597}
SPL {X  -165.650, Y  +432.479, Z    +0.000, E1   +63.557, E3 +225565.417}
SPL {X  -165.650, Y  +422.068, Z    +0.000, E1   +63.630, E3 +225575.513}
SPL {X  -165.650, Y  +409.231, Z    +0.000, E1   +63.364, E3 +225590.761}
SPL {X  -165.650, Y  +395.008, Z    +0.000, E1   +63.445, E3 +225604.524}
ENDSPLINE

SPLINE
SPL {X  -165.650, Y  +410.094, Z    +0.000, E1   +60.049, E3 +225611.974}
ENDSPLINE

SPLINE
SPL {X  -165.650, Y  +398.700, Z    +0.000, E1   +60.415, E3 +225622.872}
SPL {X  -165.650, Y  +380.643, Z    +0.000, E1   +61.187, E3 +225638.233}
SPL {X  -165.125, Y  +365.326, Z    +0.000, E1   +61.696, E3 +225651.577}
SPL {X  -164.823, Y  +361.969, Z    +0.000, E1   +60.899, E3 +225660.812}
SPL {X  -163.414, Y  +351.372, Z    +0.000, E1   +61.284, E3 +225670.074}
SPL {X  -162.189, Y  +344.818, Z    +0.000, E1   +60.900, E3 +225679.928}
SPL {X  -160.769, Y  +338.584, Z    +0.000, E1   +60.413, E3 +225690.103}
SPL {X  -157.780, Y  +328.049, Z    +0.000, E1   +60.445, E3 +225701.770}
SPL {X  -155.286, Y  +320.826, Z    +0.000, E1   +59.686, E3 +225714.326}
SPL {X  -152.445, Y  +313.689, Z    +0.000, E1   +59.490, E3 +225723.391}
SPL {X  -149.851, Y  +307.898, Z    +0.000, E1   +58.978, E3 +225732.713}
SPL {X  -146.926, Y  +301.997, Z    +0.000, E1   +58.334, E3 +225742.675}
SPL {X  -143.281, Y  +295.370, Z    +0.000, E1   +57.860, E3 +225752.443}
SPL {X  -134.010, Y  +281.128, Z    +0.000, E1   +60.923, E3 +225753.222}
SPL {X   -93.591, Y  +241.823, Z    +0.000, E1   +55.455, E3 +225845.760}
ENDSPLINE

SPLINE
SPL {X  -110.554, Y  +255.140, Z    +0.000, E1   +52.082, E3 +225972.716}
SPL {X  -137.038, Y  +285.439, Z    +0.000, E1   +46.261, E3 +225992.456}
SPL {X  -149.954, Y  +308.117, Z    +0.000, E1   +39.560, E3 +225998.803}
SPL {X  -160.070, Y  +335.868, Z    +0.000, E1   +27.320, E3 +225993.202}
SPL {X  -163.969, Y  +354.959, Z    +0.000, E1   +17.178, E3 +225993.716}
SPL {X  -165.261, Y  +367.153, Z    +0.000, E1    +9.611, E3 +225992.868}
SPL {X  -165.600, Y  +374.440, Z    +0.000, E1    +4.699, E3 +225992.130}
SPL {X  -165.650, Y  +379.657, Z    +0.000, E1    +0.819, E3 +225991.658}
SPL {X  -165.650, Y  +381.885, Z    +0.000, E1    -1.282, E3 +225990.902}
SPL {X  -165.650, Y  +386.855, Z    +0.000, E1    -7.700, E3 +225990.321}
SPL {X  -165.650, Y  +393.198, Z    +0.000, E1   -17.733, E3 +225989.297}
SPL {X  -165.650, Y  +399.991, Z    +0.000, E1   -27.922, E3 +225990.193}
SPL {X  -165.650, Y  +409.148, Z    +0.000, E1   -43.235, E3 +225985.579}
SPL {X  -165.650, Y  +420.563, Z    +0.000, E1   -54.059, E3 +225986.137}
SPL {X  -165.650, Y  +436.566, Z    +0.000, E1   -62.888, E3 +225987.850}
SPL {X  -165.650, Y  +479.770, Z    +0.000, E1   -67.621, E3 +226007.189}
SPL {X  -165.650, Y  +594.725, Z    +0.000, E1   -69.155, E3 +226074.651}
ENDSPLINE

SPLINE
SPL {X  -165.650, Y  +565.175, Z    +0.000, E1   -62.653, E3 +226098.142}
ENDSPLINE

SPLINE
SPL {X  -165.650, Y  +576.067, Z    +0.000, E1   -62.373, E3 +226111.543}
SPL {X  -165.650, Y  +586.101, Z    +0.000, E1   -62.398, E3 +226122.125}
SPL {X  -165.650, Y  +596.110, Z    +0.000, E1   -62.302, E3 +226133.566}
SPL {X  -165.650, Y  +607.052, Z    +0.000, E1   -62.387, E3 +226144.633}
SPL {X  -165.650, Y  +618.920, Z    +0.000, E1   -62.340, E3 +226157.823}
SPL {X  -165.650, Y  +631.247, Z    +0.000, E1   -62.270, E3 +226171.440}
SPL {X  -165.650, Y  +645.288, Z    +0.000, E1   -62.475, E3 +226185.120}
SPL {X  -165.650, Y  +657.265, Z    +0.000, E1   -62.410, E3 +226198.238}
SPL {X  -165.650, Y  +665.926, Z    +0.000, E1   -62.171, E3 +226209.252}
SPL {X  -165.644, Y  +676.899, Z    +0.000, E1   -62.447, E3 +226219.019}
SPL {X  -165.241, Y  +687.133, Z    +0.000, E1   -62.230, E3 +226231.722}
SPL {X  -164.056, Y  +698.425, Z    +0.000, E1   -62.113, E3 +226244.538}
SPL {X  -162.891, Y  +705.608, Z    +0.000, E1   -61.899, E3 +226253.710}
SPL {X  -160.709, Y  +715.657, Z    +0.000, E1   -61.639, E3 +226266.462}
SPL {X  -157.706, Y  +726.183, Z    +0.000, E1   -61.153, E3 +226280.845}
SPL {X  -155.057, Y  +733.785, Z    +0.000, E1   -60.834, E3 +226290.835}
SPL {X  -152.882, Y  +739.274, Z    +0.000, E1   -60.485, E3 +226298.827}
SPL {X  -150.387, Y  +744.953, Z    +0.000, E1   -60.023, E3 +226307.502}
SPL {X  -146.839, Y  +752.170, Z    +0.000, E1   -59.458, E3 +226318.461}
SPL {X  -142.415, Y  +760.104, Z    +0.000, E1   -58.730, E3 +226330.520}
SPL {X  -132.386, Y  +775.068, Z    +0.000, E1   -61.559, E3 +226332.588}
SPL {X   -89.692, Y  +814.767, Z    +0.000, E1   -54.641, E3 +226446.638}
ENDSPLINE

SPLINE
SPL {X  -120.253, Y  +789.426, Z    +0.000, E1   -51.165, E3 +226567.912}
SPL {X  -143.101, Y  +758.939, Z    +0.000, E1   -44.365, E3 +226582.020}
SPL {X  -158.740, Y  +722.846, Z    +0.000, E1   -30.140, E3 +226580.058}
SPL {X  -163.639, Y  +701.236, Z    +0.000, E1   -18.901, E3 +226582.196}
SPL {X  -165.058, Y  +689.494, Z    +0.000, E1   -11.557, E3 +226581.013}
SPL {X  -165.574, Y  +680.514, Z    +0.000, E1    -5.500, E3 +226580.257}
SPL {X  -165.650, Y  +673.883, Z    +0.000, E1    -0.454, E3 +226579.268}
SPL {X  -165.650, Y  +672.004, Z    +0.000, E1    +1.620, E3 +226578.474}
SPL {X  -165.650, Y  +669.258, Z    +0.000, E1    +5.269, E3 +226578.092}
SPL {X  -165.650, Y  +665.011, Z    +0.000, E1   +11.627, E3 +226577.979}
SPL {X  -165.650, Y  +659.446, Z    +0.000, E1   +21.123, E3 +226576.843}
SPL {X  -165.650, Y  +654.020, Z    +0.000, E1   +29.754, E3 +226576.998}
SPL {X  -165.650, Y  +644.843, Z    +0.000, E1   +43.427, E3 +226575.324}
SPL {X  -165.650, Y  +632.102, Z    +0.000, E1   +56.225, E3 +226574.673}
SPL {X  -165.650, Y  +581.672, Z    +0.000, E1   +69.744, E3 +226587.065}
SPL {X  -165.650, Y  +458.048, Z    +0.000, E1   +68.782, E3 +226667.797}
ENDSPLINE

SPLINE
SPL {X  -165.650, Y  +484.472, Z    +0.000, E1   +63.918, E3 +226682.048}
ENDSPLINE

SPLINE
SPL {X  -165.650, Y  +477.868, Z    +0.000, E1   +63.324, E3 +226693.226}
SPL {X  -165.650, Y  +463.578, Z    +0.000, E1   +63.625, E3 +226705.580}
SPL {X  -165.650, Y  +453.769, Z    +0.000, E1   +63.450, E3 +226716.838}
SPL {X  -165.650, Y  +444.234, Z    +0.000, E1   +63.262, E3 +226728.011}
SPL {X  -165.650, Y  +432.479, Z    +0.000, E1   +63.557, E3 +226737.831}
SPL {X  -165.650, Y  +422.068, Z    +0.000, E1   +63.630, E3 +226747.926}
SPL {X  -165.650, Y  +411.650, Z    +0.000, E1   +63.439, E3 +226759.945}
SPL {X  -165.650, Y  +399.089, Z    +0.000, E1   +63.334, E3 +226773.670}
ENDSPLINE

SPLINE
SPL {X  -165.650, Y  +410.094, Z    +0.000, E1   +60.049, E3 +226784.387}
ENDSPLINE

SPLINE
SPL {X  -165.650, Y  +398.700, Z    +0.000, E1   +60.415, E3 +226795.285}
SPL {X  -165.650, Y  +380.643, Z    +0.000, E1   +61.187, E3 +226810.647}
SPL {X  -165.125, Y  +365.326, Z    +0.000, E1   +61.696, E3 +226823.991}
SPL {X  -164.823, Y  +361.969, Z    +0.000, E1   +60.899, E3 +226833.226}
SPL {X  -163.414, Y  +351.372, Z    +0.000, E1   +61.284, E3 +226842.488}
SPL {X  -162.189, Y  +344.818, Z    +0.000, E1   +60.900, E3 +226852.341}
SPL {X  -160.769, Y  +338.584, Z    +0.000, E1   +60.413, E3 +226862.517}
SPL {X  -157.780, Y  +328.049, Z    +0.000, E1   +60.445, E3 +226874.184}
SPL {X  -155.286, Y  +320.826, Z    +0.000, E1   +59.686, E3 +226886.740}
SPL {X  -152.445, Y  +313.689, Z    +0.000, E1   +59.490, E3 +226895.805}
SPL {X  -149.851, Y  +307.898, Z    +0.000, E1   +58.978, E3 +226905.127}
SPL {X  -146.926, Y  +301.997, Z    +0.000, E1   +58.334, E3 +226915.089}
SPL {X  -143.997, Y  +296.618, Z    +0.000, E1   +58.069, E3 +226922.347}
SPL {X  -142.530, Y  +294.089, Z    +0.000, E1   +57.567, E3 +226927.530}
SPL {X  -134.010, Y  +281.128, Z    +0.000, E1   +60.923, E3 +226925.636}
SPL {X   -93.591, Y  +241.823, Z    +0.000, E1   +55.455, E3 +227018.174}
ENDSPLINE

SPLINE
SPL {X  -110.554, Y  +255.140, Z    +0.000, E1   +52.082, E3 +227145.130}
SPL {X  -137.038, Y  +285.439, Z    +0.000, E1   +46.261, E3 +227164.869}
SPL {X  -149.954, Y  +308.117, Z    +0.000, E1   +39.560, E3 +227171.217}
SPL {X  -160.070, Y  +335.868, Z    +0.000, E1   +27.320, E3 +227165.616}
SPL {X  -163.969, Y  +354.959, Z    +0.000, E1   +17.178, E3 +227166.130}
SPL {X  -165.261, Y  +367.153, Z    +0.000, E1    +9.611, E3 +227165.282}
SPL {X  -165.600, Y  +374.440, Z    +0.000, E1    +4.699, E3 +227164.543}
SPL {X  -165.650, Y  +379.657, Z    +0.000, E1    +0.819, E3 +227164.072}
SPL {X  -165.650, Y  +381.885, Z    +0.000, E1    -1.282, E3 +227163.316}
SPL {X  -165.650, Y  +386.855, Z    +0.000, E1    -7.700, E3 +227162.735}
SPL {X  -165.650, Y  +393.198, Z    +0.000, E1   -17.733, E3 +227161.711}
SPL {X  -165.650, Y  +399.991, Z    +0.000, E1   -27.922, E3 +227162.607}
SPL {X  -165.650, Y  +411.457, Z    +0.000, E1   -45.557, E3 +227158.355}
SPL {X  -165.650, Y  +427.627, Z    +0.000, E1   -58.747, E3 +227158.989}
SPL {X  -165.650, Y  +479.770, Z    +0.000, E1   -67.621, E3 +227179.603}
SPL {X  -165.650, Y  +594.725, Z    +0.000, E1   -69.155, E3 +227247.065}
ENDSPLINE

SPLINE
SPL {X  -165.650, Y  +565.175, Z    +0.000, E1   -62.653, E3 +227270.555}
ENDSPLINE

SPLINE
SPL {X  -165.650, Y  +576.067, Z    +0.000, E1   -62.373, E3 +227283.957}
SPL {X  -165.650, Y  +586.101, Z    +0.000, E1   -62.398, E3 +227294.539}
SPL {X  -165.650, Y  +596.110, Z    +0.000, E1   -62.302, E3 +227305.979}
SPL {X  -165.650, Y  +607.052, Z    +0.000, E1   -62.387, E3 +227317.047}
SPL {X  -165.650, Y  +615.372, Z    +0.000, E1   -62.260, E3 +227326.874}
SPL {X  -165.650, Y  +628.571, Z    +0.000, E1   -62.348, E3 +227340.594}
SPL {X  -165.650, Y  +640.498, Z    +0.000, E1   -62.343, E3 +227353.216}
SPL {X  -165.650, Y  +654.166, Z    +0.000, E1   -62.507, E3 +227366.867}
SPL {X  -165.650, Y  +665.926, Z    +0.000, E1   -62.171, E3 +227381.666}
SPL {X  -165.600, Y  +679.566, Z    +0.000, E1   -62.408, E3 +227394.703}
SPL {X  -165.066, Y  +689.394, Z    +0.000, E1   -62.143, E3 +227407.032}
SPL {X  -164.056, Y  +698.425, Z    +0.000, E1   -62.113, E3 +227416.952}
SPL {X  -162.891, Y  +705.608, Z    +0.000, E1   -61.899, E3 +227426.124}
SPL {X  -161.308, Y  +713.180, Z    +0.000, E1   -61.813, E3 +227434.818}
SPL {X  -159.339, Y  +720.787, Z    +0.000, E1   -61.452, E3 +227445.513}
SPL {X  -156.103, Y  +730.922, Z    +0.000, E1   -60.875, E3 +227460.059}
SPL {X  -152.882, Y  +739.274, Z    +0.000, E1   -60.485, E3 +227471.241}
SPL {X  -149.755, Y  +746.304, Z    +0.000, E1   -59.867, E3 +227482.362}
SPL {X  -146.068, Y  +753.629, Z    +0.000, E1   -59.384, E3 +227492.721}
SPL {X  -142.415, Y  +760.104, Z    +0.000, E1   -58.730, E3 +227502.934}
SPL {X  -132.386, Y  +775.068, Z    +0.000, E1   -61.559, E3 +227505.002}
SPL {X   -89.692, Y  +814.767, Z    +0.000, E1   -54.641, E3 +227619.051}
ENDSPLINE

SPLINE
SPL {X  -133.336, Y  +773.792, Z    +0.000, E1   -47.991, E3 +227747.518}
SPL {X  -153.017, Y  +738.949, Z    +0.000, E1   -37.928, E3 +227760.922}
SPL {X  -160.146, Y  +717.846, Z    +0.000, E1   -27.412, E3 +227748.469}
SPL {X  -163.639, Y  +701.236, Z    +0.000, E1   -18.901, E3 +227754.610}
SPL {X  -165.058, Y  +689.494, Z    +0.000, E1   -11.557, E3 +227753.427}
SPL {X  -165.574, Y  +680.514, Z    +0.000, E1    -5.500, E3 +227752.670}
SPL {X  -165.650, Y  +673.883, Z    +0.000, E1    -0.454, E3 +227751.681}
SPL {X  -165.650, Y  +672.004, Z    +0.000, E1    +1.620, E3 +227750.887}
SPL {X  -165.650, Y  +669.258, Z    +0.000, E1    +5.269, E3 +227750.506}
SPL {X  -165.650, Y  +665.011, Z    +0.000, E1   +11.627, E3 +227750.393}
SPL {X  -165.650, Y  +659.446, Z    +0.000, E1   +21.123, E3 +227749.257}
SPL {X  -165.650, Y  +654.020, Z    +0.000, E1   +29.754, E3 +227749.412}
SPL {X  -165.650, Y  +644.843, Z    +0.000, E1   +43.427, E3 +227747.738}
SPL {X  -165.650, Y  +632.102, Z    +0.000, E1   +56.225, E3 +227747.086}
SPL {X  -165.650, Y  +581.672, Z    +0.000, E1   +69.744, E3 +227759.479}
SPL {X  -165.650, Y  +458.048, Z    +0.000, E1   +68.782, E3 +227840.211}
ENDSPLINE

SPLINE
SPL {X  -165.650, Y  +484.472, Z    +0.000, E1   +63.918, E3 +227854.462}
ENDSPLINE

SPLINE
SPL {X  -165.650, Y  +477.868, Z    +0.000, E1   +63.324, E3 +227865.639}
SPL {X  -165.650, Y  +463.578, Z    +0.000, E1   +63.625, E3 +227877.993}
SPL {X  -165.650, Y  +453.769, Z    +0.000, E1   +63.450, E3 +227889.252}
SPL {X  -165.650, Y  +444.234, Z    +0.000, E1   +63.262, E3 +227900.425}
SPL {X  -165.650, Y  +432.479, Z    +0.000, E1   +63.557, E3 +227910.245}
SPL {X  -165.650, Y  +422.068, Z    +0.000, E1   +63.630, E3 +227920.340}
SPL {X  -165.650, Y  +409.231, Z    +0.000, E1   +63.364, E3 +227935.589}
SPL {X  -165.650, Y  +395.008, Z    +0.000, E1   +63.445, E3 +227949.352}
ENDSPLINE

SPLINE
SPL {X  -165.650, Y  +410.094, Z    +0.000, E1   +60.049, E3 +227956.801}
ENDSPLINE

SPLINE
SPL {X  -165.650, Y  +398.700, Z    +0.000, E1   +60.415, E3 +227967.699}
SPL {X  -165.650, Y  +380.643, Z    +0.000, E1   +61.187, E3 +227983.061}
SPL {X  -165.125, Y  +365.326, Z    +0.000, E1   +61.696, E3 +227996.404}
SPL {X  -164.823, Y  +361.969, Z    +0.000, E1   +60.899, E3 +228005.639}
SPL {X  -163.414, Y  +351.372, Z    +0.000, E1   +61.284, E3 +228014.902}
SPL {X  -162.189, Y  +344.818, Z    +0.000, E1   +60.900, E3 +228024.755}
SPL {X  -160.769, Y  +338.584, Z    +0.000, E1   +60.413, E3 +228034.931}
SPL {X  -157.780, Y  +328.049, Z    +0.000, E1   +60.445, E3 +228046.598}
SPL {X  -155.286, Y  +320.826, Z    +0.000, E1   +59.686, E3 +228059.153}
SPL {X  -152.445, Y  +313.689, Z    +0.000, E1   +59.490, E3 +228068.219}
SPL {X  -149.851, Y  +307.898, Z    +0.000, E1   +58.978, E3 +228077.541}
SPL {X  -146.926, Y  +301.997, Z    +0.000, E1   +58.334, E3 +228087.502}
SPL {X  -143.281, Y  +295.370, Z    +0.000, E1   +57.860, E3 +228097.271}
SPL {X  -134.010, Y  +281.128, Z    +0.000, E1   +60.923, E3 +228098.049}
SPL {X   -93.591, Y  +241.823, Z    +0.000, E1   +55.455, E3 +228190.587}
ENDSPLINE

SPLINE
SPL {X  -110.554, Y  +255.140, Z    +0.000, E1   +52.082, E3 +228317.543}
SPL {X  -137.038, Y  +285.439, Z    +0.000, E1   +46.261, E3 +228337.283}
SPL {X  -149.954, Y  +308.117, Z    +0.000, E1   +39.560, E3 +228343.631}
SPL {X  -160.070, Y  +335.868, Z    +0.000, E1   +27.320, E3 +228338.029}
SPL {X  -163.969, Y  +354.959, Z    +0.000, E1   +17.178, E3 +228338.544}
SPL {X  -165.261, Y  +367.153, Z    +0.000, E1    +9.611, E3 +228337.696}
SPL {X  -165.600, Y  +374.440, Z    +0.000, E1    +4.699, E3 +228336.957}
SPL {X  -165.650, Y  +380.303, Z    +0.000, E1    +0.337, E3 +228336.168}
SPL {X  -165.650, Y  +382.684, Z    +0.000, E1    -2.314, E3 +228335.662}
SPL {X  -165.650, Y  +385.555, Z    +0.000, E1    -6.051, E3 +228334.876}
SPL {X  -165.650, Y  +388.884, Z    +0.000, E1   -10.835, E3 +228335.575}
SPL {X  -165.650, Y  +393.198, Z    +0.000, E1   -17.733, E3 +228334.125}
SPL {X  -165.650, Y  +399.991, Z    +0.000, E1   -27.922, E3 +228335.021}
SPL {X  -165.650, Y  +409.148, Z    +0.000, E1   -43.235, E3 +228330.407}
SPL {X  -165.650, Y  +420.563, Z    +0.000, E1   -54.059, E3 +228330.965}
SPL {X  -165.650, Y  +436.566, Z    +0.000, E1   -62.888, E3 +228332.678}
SPL {X  -165.650, Y  +479.770, Z    +0.000, E1   -67.621, E3 +228352.016}
SPL {X  -165.650, Y  +594.725, Z    +0.000, E1   -69.155, E3 +228419.478}
ENDSPLINE

SPLINE
SPL {X  -165.650, Y  +562.482, Z    +0.000, E1   -62.785, E3 +228438.944}
ENDSPLINE

SPLINE
SPL {X  -165.650, Y  +572.898, Z    +0.000, E1   -62.409, E3 +228452.881}
SPL {X  -165.650, Y  +586.101, Z    +0.000, E1   -62.398, E3 +228466.952}
SPL {X  -165.650, Y  +596.110, Z    +0.000, E1   -62.302, E3 +228478.393}
SPL {X  -165.650, Y  +607.052, Z    +0.000, E1   -62.387, E3 +228489.460}
SPL {X  -165.650, Y  +615.372, Z    +0.000, E1   -62.260, E3 +228499.287}
SPL {X  -165.650, Y  +628.571, Z    +0.000, E1   -62.348, E3 +228513.008}
SPL {X  -165.650, Y  +645.288, Z    +0.000, E1   -62.475, E3 +228529.947}
SPL {X  -165.650, Y  +657.265, Z    +0.000, E1   -62.410, E3 +228543.066}
SPL {X  -165.650, Y  +665.926, Z    +0.000, E1   -62.171, E3 +228554.079}
SPL {X  -165.600, Y  +679.566, Z    +0.000, E1   -62.408, E3 +228567.117}
SPL {X  -165.066, Y  +689.394, Z    +0.000, E1   -62.143, E3 +228579.446}
SPL {X  -164.056, Y  +698.425, Z    +0.000, E1   -62.113, E3 +228589.366}
SPL {X  -162.891, Y  +705.608, Z    +0.000, E1   -61.899, E3 +228598.538}
SPL {X  -161.308, Y  +713.180, Z    +0.000, E1   -61.813, E3 +228607.231}
SPL {X  -159.339, Y  +720.787, Z    +0.000, E1   -61.452, E3 +228617.927}
SPL {X  -156.103, Y  +730.922, Z    +0.000, E1   -60.875, E3 +228632.473}
SPL {X  -152.882, Y  +739.274, Z    +0.000, E1   -60.485, E3 +228643.655}
SPL {X  -150.387, Y  +744.953, Z    +0.000, E1   -60.023, E3 +228652.330}
SPL {X  -146.839, Y  +752.170, Z    +0.000, E1   -59.458, E3 +228663.289}
SPL {X  -142.415, Y  +760.104, Z    +0.000, E1   -58.730, E3 +228675.347}
SPL {X  -134.606, Y  +772.046, Z    +0.000, E1   -61.105, E3 +228676.677}
SPL {X  -127.075, Y  +781.763, Z    +0.000, E1   -62.555, E3 +228678.991}
SPL {X   -89.692, Y  +814.767, Z    +0.000, E1   -54.641, E3 +228791.465}
ENDSPLINE

SPLINE
SPL {X  -133.336, Y  +773.792, Z    +0.000, E1   -47.991, E3 +228919.932}
SPL {X  -153.017, Y  +738.949, Z    +0.000, E1   -37.928, E3 +228933.336}
SPL {X  -160.146, Y  +717.846, Z    +0.000, E1   -27.412, E3 +228920.882}
SPL {X  -163.639, Y  +701.236, Z    +0.000, E1   -18.901, E3 +228927.024}
SPL {X  -165.380, Y  +684.951, Z    +0.000, E1    -8.606, E3 +228925.281}
SPL {X  -165.650, Y  +675.640, Z    +0.000, E1    -1.874, E3 +228924.817}
SPL {X  -165.650, Y  +673.425, Z    +0.000, E1    +0.051, E3 +228923.823}
SPL {X  -165.650, Y  +672.004, Z    +0.000, E1    +1.620, E3 +228923.301}
SPL {X  -165.650, Y  +669.258, Z    +0.000, E1    +5.269, E3 +228922.919}
SPL {X  -165.650, Y  +665.011, Z    +0.000, E1   +11.627, E3 +228922.807}
SPL {X  -165.650, Y  +659.446, Z    +0.000, E1   +21.123, E3 +228921.671}
SPL {X  -165.650, Y  +651.038, Z    +0.000, E1   +34.281, E3 +228921.297}
SPL {X  -165.650, Y  +635.255, Z    +0.000, E1   +53.641, E3 +228919.485}
SPL {X  -165.650, Y  +581.672, Z    +0.000, E1   +69.744, E3 +228931.892}
SPL {X  -165.650, Y  +455.882, Z    +0.000, E1   +70.075, E3 +229004.157}
ENDSPLINE

SPLINE
SPL {X  -165.650, Y  +480.501, Z    +0.000, E1   +64.561, E3 +229026.126}
ENDSPLINE

SPLINE
SPL {X  -165.650, Y  +477.868, Z    +0.000, E1   +63.324, E3 +229038.053}
SPL {X  -165.650, Y  +463.578, Z    +0.000, E1   +63.625, E3 +229050.407}
SPL {X  -165.650, Y  +453.769, Z    +0.000, E1   +63.450, E3 +229061.666}
SPL {X  -165.650, Y  +444.234, Z    +0.000, E1   +63.262, E3 +229072.839}
SPL {X  -165.650, Y  +432.479, Z    +0.000, E1   +63.557, E3 +229082.659}
SPL {X  -165.650, Y  +422.068, Z    +0.000, E1   +63.630, E3 +229092.754}
SPL {X  -165.650, Y  +411.650, Z    +0.000, E1   +63.439, E3 +229104.772}
SPL {X  -165.650, Y  +399.089, Z    +0.000, E1   +63.334, E3 +229118.498}
ENDSPLINE

SPLINE
SPL {X  -165.650, Y  +410.094, Z    +0.000, E1   +60.049, E3 +229129.215}
ENDSPLINE

SPLINE
SPL {X  -165.650, Y  +398.700, Z    +0.000, E1   +60.415, E3 +229140.113}
SPL {X  -165.650, Y  +380.643, Z    +0.000, E1   +61.187, E3 +229155.475}
SPL {X  -165.125, Y  +365.326, Z    +0.000, E1   +61.696, E3 +229168.818}
SPL {X  -164.823, Y  +361.969, Z    +0.000, E1   +60.899, E3 +229178.053}
SPL {X  -163.414, Y  +351.372, Z    +0.000, E1   +61.284, E3 +229187.316}
SPL {X  -162.189, Y  +344.818, Z    +0.000, E1   +60.900, E3 +229197.169}
SPL {X  -160.769, Y  +338.584, Z    +0.000, E1   +60.413, E3 +229207.345}
SPL {X  -158.568, Y  +330.583, Z    +0.000, E1   +60.533, E3 +229215.485}
SPL {X  -157.003, Y  +325.679, Z    +0.000, E1   +60.284, E3 +229222.455}
SPL {X  -155.286, Y  +320.826, Z    +0.000, E1   +59.686, E3 +229231.567}
SPL {X  -151.657, Y  +311.865, Z    +0.000, E1   +59.311, E3 +229243.869}
SPL {X  -147.428, Y  +302.969, Z    +0.000, E1   +58.548, E3 +229257.886}
SPL {X  -143.281, Y  +295.370, Z    +0.000, E1   +57.860, E3 +229269.684}
SPL {X  -136.453, Y  +284.583, Z    +0.000, E1   +60.257, E3 +229270.169}
SPL {X  -128.205, Y  +273.602, Z    +0.000, E1   +62.388, E3 +229270.872}
SPL {X   -93.591, Y  +241.823, Z    +0.000, E1   +55.455, E3 +229363.001}
ENDSPLINE

SPLINE
SPL {X  -110.554, Y  +255.140, Z    +0.000, E1   +52.082, E3 +229489.957}
SPL {X  -137.038, Y  +285.439, Z    +0.000, E1   +46.261, E3 +229509.697}
SPL {X  -149.954, Y  +308.117, Z    +0.000, E1   +39.560, E3 +229516.045}
SPL {X  -160.070, Y  +335.868, Z    +0.000, E1   +27.320, E3 +229510.443}
SPL {X  -163.969, Y  +354.959, Z    +0.000, E1   +17.178, E3 +229510.957}
SPL {X  -165.261, Y  +367.153, Z    +0.000, E1    +9.611, E3 +229510.110}
SPL {X  -165.600, Y  +374.440, Z    +0.000, E1    +4.699, E3 +229509.371}
SPL {X  -165.650, Y  +379.657, Z    +0.000, E1    +0.819, E3 +229508.899}
SPL {X  -165.650, Y  +381.885, Z    +0.000, E1    -1.282, E3 +229508.144}
SPL {X  -165.650, Y  +386.855, Z    +0.000, E1    -7.700, E3 +229507.563}
SPL {X  -165.650, Y  +393.198, Z    +0.000, E1   -17.733, E3 +229506.539}
SPL {X  -165.650, Y  +399.991, Z    +0.000, E1   -27.922, E3 +229507.434}
SPL {X  -165.650, Y  +411.457, Z    +0.000, E1   -45.557, E3 +229503.182}
SPL {X  -165.650, Y  +427.627, Z    +0.000, E1   -58.747, E3 +229503.816}
SPL {X  -165.650, Y  +479.770, Z    +0.000, E1   -67.621, E3 +229524.430}
SPL {X  -165.650, Y  +594.725, Z    +0.000, E1   -69.155, E3 +229591.892}
ENDSPLINE

SPLINE
SPL {X  -165.650, Y  +565.175, Z    +0.000, E1   -62.653, E3 +229615.383}
ENDSPLINE

SPLINE
SPL {X  -165.650, Y  +576.067, Z    +0.000, E1   -62.373, E3 +229628.784}
SPL {X  -165.650, Y  +586.101, Z    +0.000, E1   -62.398, E3 +229639.366}
SPL {X  -165.650, Y  +596.110, Z    +0.000, E1   -62.302, E3 +229650.807}
SPL {X  -165.650, Y  +607.052, Z    +0.000, E1   -62.387, E3 +229661.874}
SPL {X  -165.650, Y  +618.920, Z    +0.000, E1   -62.340, E3 +229675.064}
SPL {X  -165.650, Y  +631.247, Z    +0.000, E1   -62.270, E3 +229688.681}
SPL {X  -165.650, Y  +645.288, Z    +0.000, E1   -62.475, E3 +229702.361}
SPL {X  -165.650, Y  +657.265, Z    +0.000, E1   -62.410, E3 +229715.480}
SPL {X  -165.650, Y  +665.926, Z    +0.000, E1   -62.171, E3 +229726.493}
SPL {X  -165.600, Y  +679.566, Z    +0.000, E1   -62.408, E3 +229739.530}
SPL {X  -165.066, Y  +689.394, Z    +0.000, E1   -62.143, E3 +229751.860}
SPL {X  -164.056, Y  +698.425, Z    +0.000, E1   -62.113, E3 +229761.780}
SPL {X  -162.891, Y  +705.608, Z    +0.000, E1   -61.899, E3 +229770.951}
SPL {X  -161.308, Y  +713.180, Z    +0.000, E1   -61.813, E3 +229779.645}
SPL {X  -159.339, Y  +720.787, Z    +0.000, E1   -61.452, E3 +229790.340}
SPL {X  -156.103, Y  +730.922, Z    +0.000, E1   -60.875, E3 +229804.887}
SPL {X  -152.882, Y  +739.274, Z    +0.000, E1   -60.485, E3 +229816.069}
SPL {X  -149.755, Y  +746.304, Z    +0.000, E1   -59.867, E3 +229827.190}
SPL {X  -146.068, Y  +753.629, Z    +0.000, E1   -59.384, E3 +229837.549}
SPL {X  -143.119, Y  +758.908, Z    +0.000, E1   -58.828, E3 +229845.924}
SPL {X  -141.017, Y  +762.414, Z    +0.000, E1   -58.435, E3 +229851.444}
SPL {X  -132.386, Y  +775.068, Z    +0.000, E1   -61.559, E3 +229849.830}
SPL {X   -89.692, Y  +814.767, Z    +0.000, E1   -54.641, E3 +229963.879}
ENDSPLINE

SPLINE
SPL {X  -120.253, Y  +789.426, Z    +0.000, E1   -51.165, E3 +230085.153}
SPL {X  -143.101, Y  +758.939, Z    +0.000, E1   -44.365, E3 +230099.261}
SPL {X  -158.740, Y  +722.846, Z    +0.000, E1   -30.140, E3 +230097.300}
SPL {X  -163.639, Y  +701.236, Z    +0.000, E1   -18.901, E3 +230099.437}
SPL {X  -165.058, Y  +689.494, Z    +0.000, E1   -11.557, E3 +230098.254}
SPL {X  -165.574, Y  +680.514, Z    +0.000, E1    -5.500, E3 +230097.498}
SPL {X  -165.650, Y  +673.883, Z    +0.000, E1    -0.454, E3 +230096.509}
SPL {X  -165.650, Y  +672.004, Z    +0.000, E1    +1.620, E3 +230095.715}
SPL {X  -165.650, Y  +669.258, Z    +0.000, E1    +5.269, E3 +230095.333}
SPL {X  -165.650, Y  +665.011, Z    +0.000, E1   +11.627, E3 +230095.220}
SPL {X  -165.650, Y  +659.446, Z    +0.000, E1   +21.123, E3 +230094.085}
SPL {X  -165.650, Y  +654.020, Z    +0.000, E1   +29.754, E3 +230094.239}
SPL {X  -165.650, Y  +644.843, Z    +0.000, E1   +43.427, E3 +230092.565}
SPL {X  -165.650, Y  +632.102, Z    +0.000, E1   +56.225, E3 +230091.914}
SPL {X  -165.650, Y  +581.672, Z    +0.000, E1   +69.744, E3 +230104.306}
SPL {X  -165.650, Y  +458.048, Z    +0.000, E1   +68.782, E3 +230185.039}
ENDSPLINE

SPLINE
SPL {X  -165.650, Y  +484.472, Z    +0.000, E1   +63.918, E3 +230199.290}
ENDSPLINE

SPLINE
SPL {X  -165.650, Y  +477.868, Z    +0.000, E1   +63.324, E3 +230210.467}
SPL {X  -165.650, Y  +463.578, Z    +0.000, E1   +63.625, E3 +230222.821}
SPL {X  -165.650, Y  +453.769, Z    +0.000, E1   +63.450, E3 +230234.080}
SPL {X  -165.650, Y  +444.234, Z    +0.000, E1   +63.262, E3 +230245.252}
SPL {X  -165.650, Y  +432.479, Z    +0.000, E1   +63.557, E3 +230255.072}
SPL {X  -165.650, Y  +422.068, Z    +0.000, E1   +63.630, E3 +230265.168}
SPL {X  -165.650, Y  +411.650, Z    +0.000, E1   +63.439, E3 +230277.186}
SPL {X  -165.650, Y  +399.089, Z    +0.000, E1   +63.334, E3 +230290.912}
ENDSPLINE

SPLINE
SPL {X  -165.650, Y  +410.094, Z    +0.000, E1   +60.049, E3 +230301.629}
ENDSPLINE

SPLINE
SPL {X  -165.650, Y  +398.700, Z    +0.000, E1   +60.415, E3 +230312.527}
SPL {X  -165.650, Y  +380.643, Z    +0.000, E1   +61.187, E3 +230327.888}
SPL {X  -165.125, Y  +365.326, Z    +0.000, E1   +61.696, E3 +230341.232}
SPL {X  -164.823, Y  +361.969, Z    +0.000, E1   +60.899, E3 +230350.467}
SPL {X  -163.414, Y  +351.372, Z    +0.000, E1   +61.284, E3 +230359.729}
SPL {X  -162.189, Y  +344.818, Z    +0.000, E1   +60.900, E3 +230369.583}
SPL {X  -160.769, Y  +338.584, Z    +0.000, E1   +60.413, E3 +230379.759}
SPL {X  -157.780, Y  +328.049, Z    +0.000, E1   +60.445, E3 +230391.425}
SPL {X  -155.286, Y  +320.826, Z    +0.000, E1   +59.686, E3 +230403.981}
SPL {X  -152.445, Y  +313.689, Z    +0.000, E1   +59.490, E3 +230413.046}
SPL {X  -150.678, Y  +309.680, Z    +0.000, E1   +58.971, E3 +230420.358}
SPL {X  -148.010, Y  +304.117, Z    +0.000, E1   +58.696, E3 +230428.105}
SPL {X  -144.822, Y  +298.086, Z    +0.000, E1   +58.093, E3 +230437.887}
SPL {X  -142.530, Y  +294.089, Z    +0.000, E1   +57.567, E3 +230444.771}
SPL {X  -136.453, Y  +284.583, Z    +0.000, E1   +60.257, E3 +230442.582}
SPL {X  -128.205, Y  +273.602, Z    +0.000, E1   +62.388, E3 +230443.286}
SPL {X   -93.591, Y  +241.823, Z    +0.000, E1   +55.455, E3 +230535.415}
ENDSPLINE

SPLINE
SPL {X  -110.554, Y  +255.140, Z    +0.000, E1   +52.082, E3 +230662.371}
SPL {X  -137.038, Y  +285.439, Z    +0.000, E1   +46.261, E3 +230682.111}
SPL {X  -149.954, Y  +308.117, Z    +0.000, E1   +39.560, E3 +230688.458}
SPL {X  -160.070, Y  +335.868, Z    +0.000, E1   +27.320, E3 +230682.857}
SPL {X  -163.969, Y  +354.959, Z    +0.000, E1   +17.178, E3 +230683.371}
SPL {X  -165.261, Y  +367.153, Z    +0.000, E1    +9.611, E3 +230682.524}
SPL {X  -165.600, Y  +374.440, Z    +0.000, E1    +4.699, E3 +230681.785}
SPL {X  -165.650, Y  +379.657, Z    +0.000, E1    +0.819, E3 +230681.313}
SPL {X  -165.650, Y  +381.885, Z    +0.000, E1    -1.282, E3 +230680.557}
SPL {X  -165.650, Y  +386.855, Z    +0.000, E1    -7.700, E3 +230679.976}
SPL {X  -165.650, Y  +393.198, Z    +0.000, E1   -17.733, E3 +230678.952}
SPL {X  -165.650, Y  +399.991, Z    +0.000, E1   -27.922, E3 +230679.848}
SPL {X  -165.650, Y  +409.148, Z    +0.000, E1   -43.235, E3 +230675.234}
SPL {X  -165.650, Y  +420.563, Z    +0.000, E1   -54.059, E3 +230675.792}
SPL {X  -165.650, Y  +436.566, Z    +0.000, E1   -62.888, E3 +230677.505}
SPL {X  -165.650, Y  +479.770, Z    +0.000, E1   -67.621, E3 +230696.844}
SPL {X  -165.650, Y  +594.725, Z    +0.000, E1   -69.155, E3 +230764.306}
ENDSPLINE

SPLINE
SPL {X  -165.650, Y  +562.482, Z    +0.000, E1   -62.785, E3 +230783.772}
ENDSPLINE

SPLINE
SPL {X  -165.650, Y  +572.898, Z    +0.000, E1   -62.409, E3 +230797.709}
SPL {X  -165.650, Y  +586.101, Z    +0.000, E1   -62.398, E3 +230811.780}
SPL {X  -165.650, Y  +596.110, Z    +0.000, E1   -62.302, E3 +230823.221}
SPL {X  -165.650, Y  +607.052, Z    +0.000, E1   -62.387, E3 +230834.288}
SPL {X  -165.650, Y  +618.920, Z    +0.000, E1   -62.340, E3 +230847.478}
SPL {X  -165.650, Y  +631.247, Z    +0.000, E1   -62.270, E3 +230861.095}
SPL {X  -165.650, Y  +645.288, Z    +0.000, E1   -62.475, E3 +230874.775}
SPL {X  -165.650, Y  +657.265, Z    +0.000, E1   -62.410, E3 +230887.893}
SPL {X  -165.650, Y  +665.926, Z    +0.000, E1   -62.171, E3 +230898.907}
SPL {X  -165.600, Y  +679.566, Z    +0.000, E1   -62.408, E3 +230911.944}
SPL {X  -165.066, Y  +689.394, Z    +0.000, E1   -62.143, E3 +230924.273}
SPL {X  -164.056, Y  +698.425, Z    +0.000, E1   -62.113, E3 +230934.194}
SPL {X  -162.891, Y  +705.608, Z    +0.000, E1   -61.899, E3 +230943.365}
SPL {X  -161.308, Y  +713.180, Z    +0.000, E1   -61.813, E3 +230952.059}
SPL {X  -160.182, Y  +717.709, Z    +0.000, E1   -61.401, E3 +230959.671}
SPL {X  -157.706, Y  +726.183, Z    +0.000, E1   -61.153, E3 +230970.500}
SPL {X  -155.057, Y  +733.785, Z    +0.000, E1   -60.834, E3 +230980.490}
SPL {X  -152.882, Y  +739.274, Z    +0.000, E1   -60.485, E3 +230988.482}
SPL {X  -149.755, Y  +746.304, Z    +0.000, E1   -59.867, E3 +230999.604}
SPL {X  -146.068, Y  +753.629, Z    +0.000, E1   -59.384, E3 +231009.963}
SPL {X  -143.119, Y  +758.908, Z    +0.000, E1   -58.828, E3 +231018.337}
SPL {X  -141.017, Y  +762.414, Z    +0.000, E1   -58.435, E3 +231023.858}
SPL {X  -132.386, Y  +775.068, Z    +0.000, E1   -61.559, E3 +231022.244}
SPL {X   -89.692, Y  +814.767, Z    +0.000, E1   -54.641, E3 +231136.293}
ENDSPLINE

